C07229=1051.943,291.102,-104.776,172.563,37.718,157.135
C07230=1051.936,290.839,-104.743,172.560,37.714,157.134
C07231=1051.929,290.577,-104.709,172.556,37.711,157.134
C07232=1051.922,290.315,-104.675,172.553,37.708,157.133
C07233=1051.916,290.053,-104.642,172.550,37.704,157.132
C07234=1051.909,289.805,-104.611,172.546,37.701,157.131
C07235=1051.902,289.557,-104.579,172.544,37.697,157.130
C07236=1051.896,289.309,-104.547,172.540,37.694,157.130
C07237=1051.889,289.061,-104.516,172.537,37.690,157.129
C07238=1051.883,288.813,-104.484,172.534,37.687,157.128
C07239=1051.876,288.565,-104.451,172.530,37.683,157.127
C07240=1051.870,288.317,-104.420,172.528,37.680,157.126
C07241=1051.863,288.069,-104.389,172.524,37.677,157.126
C07242=1051.857,287.822,-104.358,172.522,37.673,157.125
C07243=1051.850,287.574,-104.327,172.518,37.670,157.124
C07244=1051.844,287.326,-104.295,172.516,37.667,157.123
C07245=1051.837,287.078,-104.264,172.512,37.663,157.123
C07246=1051.831,286.830,-104.232,172.509,37.660,157.122
C07247=1051.824,286.582,-104.200,172.506,37.657,157.121
C07248=1051.817,286.334,-104.169,172.503,37.653,157.120
C07249=1051.811,286.086,-104.138,172.500,37.650,157.119
C07250=1051.804,285.838,-104.106,172.497,37.647,157.119
C07251=1051.798,285.590,-104.076,172.493,37.643,157.118
C07252=1051.791,285.342,-104.044,172.491,37.640,157.117
C07253=1051.785,285.095,-104.013,172.487,37.637,157.116
C07254=1051.778,284.847,-103.982,172.485,37.634,157.116
C07255=1051.771,284.599,-103.950,172.481,37.630,157.115
C07256=1051.765,284.350,-103.919,172.479,37.627,157.114
C07257=1051.759,284.103,-103.888,172.475,37.623,157.113
C07258=1051.752,283.855,-103.857,172.472,37.620,157.113
C07259=1051.746,283.607,-103.826,172.469,37.617,157.112
C07260=1051.739,283.359,-103.795,172.466,37.613,157.111
C07261=1051.733,283.111,-103.764,172.463,37.610,157.110
C07262=1051.726,282.864,-103.732,172.460,37.606,157.109
C07263=1051.720,282.615,-103.702,172.458,37.604,157.109
C07264=1051.713,282.367,-103.670,172.454,37.600,157.108
C07265=1051.707,282.119,-103.640,172.451,37.597,157.107
C07266=1051.700,281.871,-103.608,172.448,37.593,157.106
C07267=1051.694,281.624,-103.577,172.445,37.590,157.106
C07268=1051.687,281.375,-103.546,172.442,37.587,157.105
C07269=1051.681,281.128,-103.515,172.439,37.583,157.104
C07270=1051.675,280.879,-103.484,172.437,37.580,157.103
C07271=1051.668,280.631,-103.453,172.433,37.576,157.103
C07272=1051.661,280.383,-103.422,172.430,37.574,157.102
C07273=1051.655,280.136,-103.391,172.427,37.570,157.101
C07274=1051.649,279.888,-103.360,172.424,37.567,157.100
C07275=1051.642,279.639,-103.329,172.421,37.563,157.100
C07276=1051.636,279.392,-103.298,172.418,37.560,157.099
C07277=1051.630,279.143,-103.267,172.416,37.557,157.098
C07278=1051.623,278.895,-103.237,172.412,37.553,157.097
C07279=1051.617,278.648,-103.205,172.410,37.551,157.097
C07280=1051.610,278.400,-103.175,172.406,37.547,157.096
C07281=1051.604,278.151,-103.145,172.403,37.544,157.095
C07282=1051.597,277.904,-103.114,172.401,37.541,157.094
C07283=1051.591,277.655,-103.083,172.397,37.537,157.094
C07284=1051.584,277.407,-103.051,172.395,37.534,157.093
C07285=1051.578,277.160,-103.022,172.391,37.531,157.092
C07286=1051.571,276.909,-102.990,172.389,37.527,157.091
C07287=1051.565,276.657,-102.960,172.386,37.524,157.091
C07288=1051.558,276.407,-102.928,172.382,37.520,157.090
C07289=1051.551,276.156,-102.898,172.380,37.518,157.089
C07290=1051.545,275.908,-102.867,172.377,37.514,157.088
C07291=1051.539,275.660,-102.836,172.374,37.511,157.088
C07292=1051.533,275.412,-102.805,172.371,37.508,157.087
C07293=1051.526,275.164,-102.775,172.368,37.504,157.086
C07294=1051.519,274.916,-102.745,172.365,37.501,157.085
C07295=1051.513,274.668,-102.714,172.363,37.498,157.085
C07296=1051.507,274.419,-102.684,172.359,37.494,157.084
C07297=1051.500,274.172,-102.653,172.357,37.491,157.083
C07298=1051.494,273.924,-102.622,172.354,37.488,157.082
C07299=1051.487,273.675,-102.592,172.350,37.485,157.082
C07300=1051.481,273.428,-102.562,172.348,37.482,157.081
C07301=1051.474,273.179,-102.531,172.345,37.478,157.080
C07302=1051.468,272.932,-102.501,172.342,37.475,157.079
C07303=1051.461,272.683,-102.471,172.339,37.472,157.079
C07304=1051.455,272.436,-102.440,172.337,37.468,157.078
C07305=1051.449,272.187,-102.410,172.333,37.465,157.077
C07306=1051.442,271.939,-102.380,172.331,37.462,157.077
C07307=1051.436,271.691,-102.349,172.328,37.458,157.076
C07308=1051.429,271.443,-102.319,172.325,37.456,157.075
C07309=1051.423,271.195,-102.289,172.322,37.452,157.074
C07310=1051.416,270.947,-102.259,172.320,37.449,157.074
C07311=1051.410,270.699,-102.228,172.317,37.446,157.073
C07312=1051.403,270.451,-102.198,172.313,37.442,157.072
C07313=1051.397,270.203,-102.168,172.311,37.439,157.071
C07314=1051.390,269.955,-102.138,172.308,37.436,157.071
C07315=1051.384,269.707,-102.107,172.305,37.433,157.070
C07316=1051.377,269.459,-102.077,172.302,37.429,157.069
C07317=1051.371,269.210,-102.048,172.300,37.427,157.069
C07318=1051.364,268.962,-102.017,172.297,37.423,157.068
C07319=1051.358,268.714,-101.987,172.294,37.420,157.067
C07320=1051.352,268.467,-101.957,172.291,37.417,157.066
C07321=1051.346,268.218,-101.927,172.289,37.413,157.066
C07322=1051.339,267.970,-101.898,172.285,37.410,157.065
C07323=1051.332,267.722,-101.867,172.283,37.407,157.064
C07324=1051.326,267.474,-101.837,172.280,37.404,157.064
C07325=1051.319,267.226,-101.807,172.278,37.400,157.063
C07326=1051.314,266.977,-101.777,172.274,37.398,157.062
C07327=1051.306,266.729,-101.747,172.272,37.394,157.061
C07328=1051.300,266.482,-101.717,172.269,37.391,157.061
C07329=1051.294,266.232,-101.687,172.267,37.388,157.060
C07330=1051.287,265.985,-101.658,172.263,37.385,157.059
C07331=1051.281,265.737,-101.628,172.261,37.381,157.058
C07332=1051.275,265.488,-101.598,172.258,37.378,157.058
C07333=1051.268,265.241,-101.568,172.256,37.375,157.057
C07334=1051.261,264.993,-101.538,172.252,37.372,157.056
C07335=1051.255,264.744,-101.508,172.250,37.368,157.056
C07336=1051.249,264.497,-101.479,172.247,37.365,157.055
C07337=1051.242,264.248,-101.449,172.244,37.362,157.054
C07338=1051.236,264.001,-101.420,172.242,37.359,157.053
C07339=1051.229,263.753,-101.390,172.238,37.356,157.053
C07340=1051.223,263.506,-101.360,172.236,37.352,157.052
C07341=1051.216,263.258,-101.331,172.233,37.349,157.051
C07342=1051.210,263.012,-101.301,172.231,37.346,157.050
C07343=1051.204,262.764,-101.271,172.228,37.343,157.050
C07344=1051.197,262.517,-101.242,172.225,37.340,157.049
C07345=1051.191,262.269,-101.212,172.222,37.336,157.048
C07346=1051.184,262.021,-101.183,172.220,37.333,157.048
C07347=1051.178,261.772,-101.154,172.217,37.330,157.047
C07348=1051.171,261.525,-101.124,172.215,37.327,157.046
C07349=1051.165,261.277,-101.095,172.211,37.324,157.046
C07350=1051.158,261.028,-101.065,172.209,37.321,157.045
C07351=1051.151,260.780,-101.036,172.206,37.318,157.044
C07352=1051.145,260.532,-101.007,172.204,37.315,157.044
C07353=1051.138,260.283,-100.977,172.201,37.311,157.043
C07354=1051.132,260.036,-100.947,172.198,37.308,157.042
C07355=1051.125,259.787,-100.918,172.196,37.305,157.042
C07356=1051.119,259.539,-100.889,172.193,37.302,157.041
C07357=1051.112,259.291,-100.859,172.191,37.299,157.040
C07358=1051.105,259.042,-100.830,172.188,37.295,157.039
C07359=1051.099,258.794,-100.801,172.184,37.293,157.039
C07360=1051.093,258.546,-100.772,172.182,37.290,157.038
C07361=1051.086,258.298,-100.743,172.179,37.286,157.037
C07362=1051.079,258.050,-100.713,172.177,37.283,157.037
C07363=1051.072,257.802,-100.684,172.175,37.280,157.036
C07364=1051.066,257.554,-100.655,172.172,37.277,157.035
C07365=1051.059,257.305,-100.626,172.170,37.274,157.035
C07366=1051.053,257.057,-100.597,172.166,37.270,157.034
C07367=1051.047,256.809,-100.568,172.164,37.267,157.033
C07368=1051.040,256.561,-100.538,172.161,37.264,157.032
C07369=1051.033,256.312,-100.508,172.159,37.261,157.032
C07370=1051.027,256.064,-100.479,172.156,37.258,157.031
C07371=1051.021,255.816,-100.450,172.154,37.255,157.030
C07372=1051.015,255.568,-100.421,172.151,37.252,157.030
C07373=1051.008,255.319,-100.392,172.148,37.249,157.029
C07374=1051.001,255.071,-100.363,172.145,37.245,157.028
C07375=1050.995,254.823,-100.334,172.143,37.242,157.028
C07376=1050.988,254.575,-100.305,172.140,37.239,157.027
C07377=1050.982,254.327,-100.276,172.138,37.236,157.026
C07378=1050.976,254.093,-100.249,172.135,37.233,157.026
C07379=1050.970,253.860,-100.221,172.133,37.230,157.025
C07380=1050.964,253.626,-100.194,172.130,37.227,157.024
C07381=1050.958,253.392,-100.167,172.128,37.223,157.023
C07382=1050.952,253.158,-100.139,172.125,37.221,157.023
C07383=1050.946,252.925,-100.112,172.123,37.218,157.022
C07384=1050.940,252.692,-100.085,172.120,37.215,157.022
C07385=1050.934,252.458,-100.057,172.118,37.212,157.021
C07386=1050.928,252.210,-100.028,172.116,37.209,157.020
C07387=1050.920,251.962,-99.999,172.113,37.205,157.019
C07388=1050.914,251.713,-99.971,172.111,37.202,157.019
C07389=1050.908,251.465,-99.942,172.108,37.199,157.018
C07390=1050.902,251.217,-99.913,172.106,37.196,157.017
C07391=1050.896,250.969,-99.884,172.103,37.192,157.017
C07392=1050.889,250.720,-99.855,172.101,37.189,157.016
C07393=1050.883,250.472,-99.826,172.098,37.186,157.015
C07394=1050.877,250.224,-99.797,172.096,37.183,157.015
C07395=1050.871,249.975,-99.768,172.093,37.180,157.014
C07396=1050.864,249.728,-99.740,172.091,37.176,157.013
C07397=1050.858,249.479,-99.711,172.088,37.174,157.013
C07398=1050.851,249.201,-99.678,172.085,37.169,157.012
C07399=1050.843,248.924,-99.646,172.082,37.166,157.011
C07400=1050.837,248.646,-99.614,172.079,37.162,157.010
C07401=1050.830,248.368,-99.582,172.077,37.159,157.009
C07402=1050.823,248.121,-99.553,172.075,37.156,157.009
C07403=1050.817,247.872,-99.525,172.072,37.152,157.008
C07404=1050.810,247.624,-99.496,172.070,37.149,157.007
C07405=1050.804,247.376,-99.467,172.067,37.146,157.006
C07406=1050.798,247.127,-99.438,172.065,37.143,157.006
C07407=1050.792,246.879,-99.409,172.062,37.139,157.005
C07408=1050.786,246.631,-99.380,172.060,37.136,157.004
C07409=1050.779,246.382,-99.353,172.057,37.133,157.004
C07410=1050.773,246.134,-99.323,172.055,37.130,157.003
C07411=1050.767,245.886,-99.294,172.052,37.126,157.002
C07412=1050.761,245.637,-99.266,172.050,37.123,157.002
C07413=1050.754,245.389,-99.238,172.047,37.120,157.001
C07414=1050.748,245.141,-99.209,172.045,37.117,157.000
C07415=1050.741,244.892,-99.180,172.042,37.114,157.000
C07416=1050.735,244.644,-99.153,172.040,37.111,156.999
C07417=1050.729,244.396,-99.124,172.037,37.108,156.998
C07418=1050.722,244.147,-99.096,172.035,37.104,156.997
C07419=1050.716,243.899,-99.067,172.032,37.101,156.997
C07420=1050.710,243.651,-99.038,172.030,37.098,156.996
C07421=1050.703,243.403,-99.010,172.027,37.095,156.995
C07422=1050.697,243.155,-98.982,172.025,37.092,156.995
C07423=1050.690,242.907,-98.954,172.022,37.088,156.994
C07424=1050.684,242.658,-98.925,172.020,37.085,156.993
C07425=1050.678,242.409,-98.897,172.017,37.082,156.993
C07426=1050.671,242.162,-98.869,172.015,37.079,156.992
C07427=1050.666,241.913,-98.840,172.013,37.076,156.991
C07428=1050.659,241.665,-98.812,172.010,37.072,156.990
C07429=1050.653,241.416,-98.783,172.008,37.069,156.990
C07430=1050.646,241.168,-98.756,172.005,37.066,156.989
C07431=1050.639,240.920,-98.727,172.003,37.063,156.988
C07432=1050.633,240.671,-98.699,172.000,37.060,156.988
C07433=1050.626,240.423,-98.671,171.999,37.056,156.987
C07434=1050.620,240.174,-98.643,171.996,37.053,156.986
C07435=1050.613,239.926,-98.614,171.994,37.050,156.986
C07436=1050.607,239.678,-98.587,171.991,37.047,156.985
C07437=1050.601,239.429,-98.558,171.989,37.044,156.984
C07438=1050.595,239.181,-98.531,171.987,37.041,156.984
C07439=1050.588,238.933,-98.503,171.984,37.037,156.983
C07440=1050.582,238.685,-98.474,171.982,37.034,156.982
C07441=1050.575,238.436,-98.446,171.979,37.031,156.982
C07442=1050.568,238.188,-98.419,171.977,37.028,156.981
C07443=1050.562,237.939,-98.390,171.974,37.025,156.980
C07444=1050.556,237.691,-98.363,171.972,37.021,156.980
C07445=1050.549,237.442,-98.335,171.969,37.018,156.979
C07446=1050.542,237.194,-98.307,171.968,37.015,156.978
C07447=1050.537,236.946,-98.279,171.965,37.012,156.977
C07448=1050.530,236.698,-98.251,171.963,37.009,156.977
C07449=1050.523,236.449,-98.223,171.961,37.006,156.976
C07450=1050.517,236.201,-98.195,171.958,37.002,156.975
C07451=1050.511,235.952,-98.167,171.956,36.999,156.975
C07452=1050.504,235.704,-98.139,171.953,36.996,156.974
C07453=1050.497,235.455,-98.112,171.951,36.993,156.973
C07454=1050.491,235.201,-98.083,171.948,36.990,156.973
C07455=1050.485,234.947,-98.055,171.946,36.986,156.972
C07456=1050.478,234.694,-98.026,171.944,36.983,156.971
C07457=1050.472,234.439,-97.997,171.942,36.980,156.971
C07458=1050.465,234.191,-97.970,171.939,36.977,156.970
C07459=1050.459,233.943,-97.942,171.937,36.973,156.969
C07460=1050.453,233.694,-97.914,171.934,36.970,156.969
C07461=1050.447,233.446,-97.886,171.932,36.967,156.968
C07462=1050.440,233.198,-97.859,171.930,36.964,156.967
C07463=1050.433,232.949,-97.831,171.928,36.960,156.966
C07464=1050.427,232.700,-97.804,171.926,36.957,156.966
C07465=1050.422,232.452,-97.776,171.923,36.954,156.965
C07466=1050.415,232.204,-97.748,171.921,36.951,156.964
C07467=1050.408,231.955,-97.720,171.918,36.948,156.964
C07468=1050.402,231.707,-97.693,171.916,36.944,156.963
C07469=1050.395,231.458,-97.665,171.913,36.941,156.962
C07470=1050.389,231.211,-97.638,171.912,36.938,156.962
C07471=1050.383,230.962,-97.611,171.909,36.935,156.961
C07472=1050.377,230.713,-97.582,171.907,36.932,156.960
C07473=1050.371,230.465,-97.555,171.904,36.928,156.960
C07474=1050.364,230.217,-97.527,171.902,36.925,156.959
C07475=1050.357,229.968,-97.499,171.901,36.922,156.958
C07476=1050.351,229.719,-97.472,171.898,36.919,156.958
C07477=1050.345,229.471,-97.445,171.896,36.916,156.957
C07478=1050.338,229.223,-97.417,171.893,36.912,156.956
C07479=1050.331,228.974,-97.390,171.891,36.909,156.956
C07480=1050.325,228.725,-97.363,171.889,36.906,156.955
C07481=1050.319,228.478,-97.335,171.887,36.903,156.954
C07482=1050.312,228.229,-97.307,171.885,36.900,156.954
C07483=1050.306,227.980,-97.280,171.882,36.897,156.953
C07484=1050.300,227.732,-97.253,171.880,36.893,156.952
C07485=1050.293,227.483,-97.226,171.877,36.890,156.951
C07486=1050.286,227.235,-97.199,171.876,36.887,156.951
C07487=1050.279,226.987,-97.171,171.873,36.884,156.950
C07488=1050.273,226.738,-97.145,171.871,36.881,156.949
C07489=1050.267,226.490,-97.117,171.868,36.877,156.949
C07490=1050.260,226.241,-97.090,171.867,36.874,156.948
C07491=1050.254,225.993,-97.062,171.865,36.871,156.947
C07492=1050.248,225.745,-97.035,171.862,36.868,156.947
C07493=1050.241,225.496,-97.008,171.860,36.865,156.946
C07494=1050.235,225.248,-96.980,171.857,36.862,156.945
C07495=1050.228,224.999,-96.954,171.856,36.858,156.945
C07496=1050.221,224.751,-96.926,171.853,36.855,156.944
C07497=1050.216,224.502,-96.900,171.851,36.852,156.943
C07498=1050.209,224.254,-96.872,171.848,36.849,156.943
C07499=1050.203,224.006,-96.845,171.847,36.846,156.942
C07500=1050.197,223.757,-96.817,171.845,36.842,156.941
C07501=1050.190,223.508,-96.790,171.842,36.839,156.941
C07502=1050.184,223.260,-96.764,171.840,36.836,156.940
C07503=1050.177,223.012,-96.737,171.838,36.833,156.939
C07504=1050.171,222.763,-96.710,171.836,36.829,156.939
C07505=1050.164,222.515,-96.682,171.833,36.826,156.938
C07506=1050.158,222.266,-96.655,171.831,36.823,156.937
C07507=1050.152,222.018,-96.628,171.830,36.819,156.937
C07508=1050.146,221.769,-96.601,171.827,36.816,156.936
C07509=1050.139,221.521,-96.575,171.825,36.813,156.935
C07510=1050.132,221.259,-96.545,171.823,36.809,156.934
C07511=1050.126,220.997,-96.517,171.821,36.806,156.934
C07512=1050.119,220.736,-96.489,171.818,36.803,156.933
C07513=1050.113,220.474,-96.460,171.816,36.799,156.932
C07514=1050.105,220.226,-96.433,171.813,36.796,156.932
C07515=1050.099,219.977,-96.407,171.812,36.793,156.931
C07516=1050.092,219.729,-96.380,171.809,36.790,156.930
C07517=1050.087,219.480,-96.354,171.807,36.787,156.930
C07518=1050.080,219.232,-96.326,171.806,36.783,156.929
C07519=1050.073,218.984,-96.300,171.803,36.780,156.928
C07520=1050.067,218.735,-96.273,171.801,36.777,156.927
C07521=1050.060,218.486,-96.246,171.798,36.774,156.927
C07522=1050.054,218.238,-96.220,171.797,36.771,156.926
C07523=1050.047,217.989,-96.192,171.794,36.767,156.925
C07524=1050.041,217.741,-96.166,171.792,36.764,156.925
C07525=1050.035,217.492,-96.139,171.791,36.760,156.924
C07526=1050.028,217.244,-96.113,171.788,36.757,156.923
C07527=1050.022,216.995,-96.086,171.786,36.754,156.923
C07528=1050.015,216.747,-96.060,171.784,36.751,156.922
C07529=1050.009,216.498,-96.033,171.782,36.748,156.921
C07530=1050.003,216.250,-96.005,171.779,36.744,156.921
C07531=1049.996,216.001,-95.979,171.778,36.741,156.920
C07532=1049.990,215.753,-95.952,171.776,36.738,156.919
C07533=1049.983,215.504,-95.926,171.773,36.735,156.919
C07534=1049.977,215.256,-95.899,171.772,36.731,156.918
C07535=1049.970,215.007,-95.873,171.769,36.728,156.917
C07536=1049.964,214.759,-95.846,171.767,36.725,156.917
C07537=1049.958,214.510,-95.820,171.765,36.722,156.916
C07538=1049.951,214.262,-95.793,171.763,36.719,156.915
C07539=1049.945,214.013,-95.767,171.761,36.715,156.915
C07540=1049.938,213.765,-95.740,171.759,36.712,156.914
C07541=1049.932,213.516,-95.713,171.757,36.708,156.913
C07542=1049.925,213.267,-95.687,171.755,36.705,156.913
C07543=1049.920,213.019,-95.660,171.753,36.702,156.912
C07544=1049.913,212.771,-95.634,171.750,36.699,156.911
C07545=1049.907,212.522,-95.607,171.749,36.695,156.910
C07546=1049.900,212.274,-95.581,171.747,36.692,156.910
C07547=1049.894,212.025,-95.554,171.744,36.689,156.909
C07548=1049.887,211.777,-95.528,171.743,36.686,156.908
C07549=1049.881,211.528,-95.501,171.740,36.682,156.908
C07550=1049.874,211.280,-95.475,171.739,36.679,156.907
C07551=1049.868,211.031,-95.450,171.736,36.675,156.906
C07552=1049.862,210.782,-95.423,171.734,36.672,156.906
C07553=1049.855,210.534,-95.397,171.733,36.669,156.905
C07554=1049.849,210.285,-95.370,171.730,36.666,156.904
C07555=1049.842,210.037,-95.344,171.729,36.662,156.904
C07556=1049.836,209.789,-95.318,171.726,36.659,156.903
C07557=1049.830,209.539,-95.291,171.724,36.656,156.902
C07558=1049.823,209.291,-95.265,171.723,36.653,156.902
C07559=1049.817,209.043,-95.239,171.720,36.649,156.901
C07560=1049.810,208.794,-95.212,171.719,36.646,156.900
C07561=1049.804,208.546,-95.186,171.716,36.643,156.899
C07562=1049.797,208.297,-95.160,171.714,36.640,156.899
C07563=1049.791,208.049,-95.134,171.712,36.636,156.898
C07564=1049.785,207.800,-95.108,171.710,36.633,156.897
C07565=1049.778,207.551,-95.081,171.709,36.629,156.897
C07566=1049.771,207.295,-95.055,171.706,36.626,156.896
C07567=1049.765,207.039,-95.028,171.704,36.623,156.895
C07568=1049.758,206.783,-95.001,171.702,36.619,156.895
C07569=1049.752,206.527,-94.974,171.700,36.616,156.894
C07570=1049.726,205.475,-94.869,171.467,36.519,156.874
C07571=1049.720,205.226,-94.843,171.464,36.516,156.873
C07572=1049.714,204.977,-94.818,171.462,36.514,156.873
C07573=1049.707,204.729,-94.793,171.460,36.512,156.872
C07574=1049.702,204.480,-94.768,171.457,36.509,156.872
C07575=1049.695,204.232,-94.744,171.454,36.507,156.871
C07576=1049.689,203.983,-94.718,171.452,36.504,156.871
C07577=1049.683,203.734,-94.694,171.449,36.501,156.870
C07578=1049.677,203.485,-94.668,171.446,36.499,156.870
C07579=1049.671,203.237,-94.643,171.444,36.497,156.869
C07580=1049.665,202.988,-94.619,171.442,36.494,156.869
C07581=1049.659,202.739,-94.593,171.438,36.492,156.868
C07582=1049.654,202.491,-94.568,171.436,36.489,156.868
C07583=1049.648,202.242,-94.544,171.434,36.487,156.867
C07584=1049.641,201.993,-94.518,171.431,36.484,156.867
C07585=1049.636,201.744,-94.494,171.428,36.482,156.866
C07586=1049.629,201.496,-94.469,171.426,36.480,156.866
C07587=1049.623,201.247,-94.445,171.424,36.477,156.865
C07588=1049.617,200.998,-94.419,171.420,36.475,156.865
C07589=1049.610,200.749,-94.395,171.418,36.472,156.864
C07590=1049.604,200.501,-94.370,171.416,36.470,156.864
C07591=1049.599,200.252,-94.346,171.413,36.467,156.863
C07592=1049.592,200.004,-94.321,171.410,36.465,156.863
C07593=1049.586,199.755,-94.296,171.408,36.463,156.862
C07594=1049.579,199.506,-94.272,171.406,36.460,156.862
C07595=1049.574,199.258,-94.247,171.403,36.458,156.861
C07596=1049.567,199.009,-94.223,171.400,36.456,156.861
C07597=1049.561,198.760,-94.198,171.398,36.454,156.861
C07598=1049.556,198.511,-94.174,171.396,36.451,156.860
C07599=1049.549,198.263,-94.149,171.392,36.449,156.860
C07600=1049.543,198.014,-94.125,171.390,36.446,156.859
C07601=1049.537,197.765,-94.101,171.388,36.444,156.859
C07602=1049.531,197.517,-94.076,171.385,36.441,156.858
C07603=1049.525,197.267,-94.051,171.383,36.439,156.858
C07604=1049.518,197.018,-94.027,171.380,36.437,156.857
C07605=1049.512,196.771,-94.002,171.378,36.435,156.857
C07606=1049.506,196.522,-93.978,171.375,36.432,156.856
C07607=1049.501,196.273,-93.954,171.373,36.430,156.856
C07608=1049.494,196.025,-93.929,171.370,36.427,156.855
C07609=1049.488,195.775,-93.904,171.367,36.425,156.855
C07610=1049.482,195.527,-93.881,171.365,36.423,156.854
C07611=1049.476,195.278,-93.856,171.363,36.421,156.854
C07612=1049.470,195.029,-93.831,171.361,36.418,156.853
C07613=1049.464,194.781,-93.807,171.357,36.416,156.853
C07614=1049.458,194.532,-93.782,171.355,36.413,156.852
C07615=1049.452,194.283,-93.759,171.353,36.411,156.852
C07616=1049.446,194.034,-93.734,171.351,36.409,156.851
C07617=1049.439,193.786,-93.709,171.348,36.407,156.851
C07618=1049.433,193.537,-93.685,171.345,36.404,156.851
C07619=1049.427,193.288,-93.661,171.343,36.402,156.850
C07620=1049.422,193.039,-93.637,171.340,36.399,156.850
C07621=1049.415,192.790,-93.613,171.338,36.397,156.849
C07622=1049.410,192.542,-93.588,171.336,36.395,156.849
C07623=1049.403,192.293,-93.564,171.333,36.393,156.848
C07624=1049.397,192.044,-93.539,171.330,36.390,156.848
C07625=1049.391,191.796,-93.515,171.328,36.388,156.847
C07626=1049.385,191.547,-93.491,171.326,36.385,156.847
C07627=1049.379,191.298,-93.467,171.324,36.384,156.846
C07628=1049.373,191.049,-93.443,171.321,36.381,156.846
C07629=1049.368,190.801,-93.418,171.318,36.379,156.846
C07630=1049.361,190.552,-93.394,171.316,36.376,156.845
C07631=1049.354,190.267,-93.367,171.314,36.374,156.845
C07632=1049.347,189.983,-93.339,171.310,36.371,156.844
C07633=1049.341,189.699,-93.312,171.308,36.368,156.843
C07634=1049.334,189.414,-93.284,171.305,36.366,156.843
C07635=1049.328,189.166,-93.260,171.302,36.364,156.842
C07636=1049.322,188.917,-93.235,171.300,36.361,156.842
C07637=1049.316,188.669,-93.212,171.298,36.359,156.842
C07638=1049.310,188.419,-93.187,171.296,36.357,156.841
C07639=1049.304,188.171,-93.163,171.293,36.354,156.841
C07640=1049.299,187.921,-93.139,171.291,36.352,156.840
C07641=1049.292,187.673,-93.116,171.289,36.350,156.840
C07642=1049.287,187.424,-93.091,171.286,36.348,156.839
C07643=1049.281,187.175,-93.067,171.283,36.345,156.839
C07644=1049.275,186.927,-93.043,171.281,36.343,156.838
C07645=1049.269,186.678,-93.019,171.279,36.340,156.838
C07646=1049.263,186.429,-92.995,171.276,36.339,156.837
C07647=1049.257,186.180,-92.971,171.274,36.336,156.837
C07648=1049.251,185.932,-92.947,171.272,36.334,156.836
C07649=1049.246,185.683,-92.924,171.270,36.331,156.836
C07650=1049.239,185.434,-92.900,171.267,36.329,156.836
C07651=1049.234,185.185,-92.875,171.264,36.327,156.835
C07652=1049.228,184.937,-92.852,171.262,36.324,156.835
C07653=1049.222,184.688,-92.827,171.260,36.322,156.834
C07654=1049.216,184.439,-92.803,171.257,36.320,156.834
C07655=1049.211,184.190,-92.780,171.255,36.318,156.833
C07656=1049.204,183.941,-92.756,171.253,36.315,156.833
C07657=1049.198,183.693,-92.732,171.251,36.313,156.832
C07658=1049.192,183.443,-92.709,171.248,36.311,156.832
C07659=1049.186,183.195,-92.685,171.246,36.309,156.832
C07660=1049.179,182.946,-92.661,171.244,36.307,156.831
C07661=1049.173,182.697,-92.638,171.241,36.305,156.831
C07662=1049.167,182.448,-92.614,171.238,36.303,156.830
C07663=1049.161,182.199,-92.591,171.236,36.301,156.830
C07664=1049.155,181.951,-92.568,171.234,36.299,156.830
C07665=1049.148,181.702,-92.544,171.232,36.296,156.829
C07666=1049.143,181.453,-92.521,171.230,36.295,156.829
C07667=1049.135,181.204,-92.497,171.227,36.292,156.828
C07668=1049.129,180.956,-92.474,171.225,36.290,156.828
C07669=1049.123,180.707,-92.450,171.223,36.288,156.828
C07670=1049.117,180.458,-92.427,171.220,36.286,156.827
C07671=1049.111,180.209,-92.404,171.217,36.284,156.827
C07672=1049.105,179.960,-92.380,171.215,36.282,156.826
C07673=1049.099,179.711,-92.357,171.213,36.280,156.826
C07674=1049.093,179.463,-92.334,171.211,36.277,156.825
C07675=1049.086,179.214,-92.310,171.208,36.276,156.825
C07676=1049.081,178.965,-92.287,171.206,36.274,156.825
C07677=1049.074,178.716,-92.263,171.204,36.271,156.824
C07678=1049.068,178.467,-92.240,171.202,36.269,156.824
C07679=1049.062,178.219,-92.216,171.199,36.267,156.823
C07680=1049.055,177.969,-92.193,171.197,36.265,156.823
C07681=1049.049,177.720,-92.170,171.195,36.263,156.822
C07682=1049.043,177.472,-92.147,171.192,36.261,156.822
C07683=1049.038,177.223,-92.124,171.190,36.259,156.822
C07684=1049.031,176.974,-92.100,171.187,36.257,156.821
C07685=1049.025,176.725,-92.077,171.185,36.255,156.821
C07686=1049.020,176.476,-92.054,171.183,36.252,156.820
C07687=1049.013,176.227,-92.030,171.181,36.250,156.820
C07688=1049.007,175.979,-92.007,171.178,36.249,156.820
C07689=1049.000,175.731,-91.984,171.176,36.246,156.819
C07690=1048.994,175.481,-91.961,171.174,36.244,156.819
C07691=1048.988,175.232,-91.938,171.172,36.242,156.818
C07692=1048.983,174.983,-91.915,171.170,36.240,156.818
C07693=1048.977,174.735,-91.891,171.167,36.238,156.818
C07694=1048.970,174.485,-91.868,171.165,36.236,156.817
C07695=1048.963,174.201,-91.842,171.163,36.233,156.817
C07696=1048.956,173.916,-91.815,171.160,36.231,156.816
C07697=1048.950,173.631,-91.788,171.157,36.229,156.816
C07698=1048.942,173.347,-91.762,171.155,36.226,156.815
C07699=1048.937,173.098,-91.739,171.153,36.224,156.815
C07700=1048.931,172.849,-91.716,171.151,36.222,156.814
C07701=1048.925,172.600,-91.693,171.148,36.220,156.814
C07702=1048.918,172.351,-91.669,171.146,36.218,156.814
C07703=1048.912,172.102,-91.646,171.144,36.216,156.813
C07704=1048.906,171.854,-91.623,171.142,36.214,156.813
C07705=1048.901,171.605,-91.601,171.139,36.212,156.812
C07706=1048.895,171.356,-91.578,171.137,36.210,156.812
C07707=1048.889,171.107,-91.555,171.135,36.207,156.812
C07708=1048.882,170.858,-91.531,171.133,36.206,156.811
C07709=1048.876,170.609,-91.508,171.131,36.203,156.811
C07710=1048.870,170.360,-91.485,171.128,36.201,156.810
C07711=1048.865,170.112,-91.462,171.126,36.199,156.810
C07712=1048.859,169.863,-91.439,171.124,36.197,156.810
C07713=1048.853,169.614,-91.416,171.122,36.195,156.809
C07714=1048.847,169.365,-91.394,171.119,36.193,156.809
C07715=1048.840,169.116,-91.371,171.117,36.191,156.808
C07716=1048.834,168.867,-91.347,171.115,36.189,156.808
C07717=1048.829,168.618,-91.324,171.113,36.187,156.807
C07718=1048.823,168.369,-91.301,171.111,36.185,156.807
C07719=1048.817,168.121,-91.278,171.108,36.183,156.807
C07720=1048.811,167.872,-91.255,171.106,36.180,156.806
C07721=1048.805,167.623,-91.233,171.104,36.179,156.806
C07722=1048.799,167.374,-91.210,171.102,36.176,156.805
C07723=1048.793,167.125,-91.187,171.099,36.174,156.805
C07724=1048.788,166.876,-91.164,171.097,36.172,156.805
C07725=1048.782,166.627,-91.141,171.095,36.170,156.804
C07726=1048.775,166.379,-91.119,171.093,36.168,156.804
C07727=1048.769,166.129,-91.096,171.091,36.166,156.804
C07728=1048.763,165.880,-91.073,171.088,36.164,156.803
C07729=1048.758,165.632,-91.050,171.086,36.162,156.803
C07730=1048.752,165.383,-91.027,171.084,36.159,156.802
C07731=1048.745,165.134,-91.004,171.082,36.158,156.802
C07732=1048.740,164.885,-90.981,171.079,36.156,156.801
C07733=1048.734,164.636,-90.959,171.077,36.153,156.801
C07734=1048.729,164.387,-90.936,171.076,36.151,156.801
C07735=1048.723,164.138,-90.913,171.074,36.150,156.800
C07736=1048.716,163.889,-90.891,171.072,36.147,156.800
C07737=1048.711,163.640,-90.868,171.069,36.145,156.799
C07738=1048.705,163.391,-90.845,171.067,36.143,156.799
C07739=1048.699,163.143,-90.822,171.065,36.141,156.799
C07740=1048.693,162.894,-90.800,171.063,36.139,156.798
C07741=1048.687,162.644,-90.778,171.060,36.137,156.798
C07742=1048.682,162.396,-90.755,171.058,36.135,156.797
C07743=1048.676,162.147,-90.732,171.056,36.133,156.797
C07744=1048.669,161.898,-90.709,171.054,36.130,156.797
C07745=1048.664,161.650,-90.687,171.053,36.129,156.796
C07746=1048.658,161.401,-90.664,171.050,36.127,156.796
C07747=1048.653,161.151,-90.642,171.048,36.124,156.795
C07748=1048.647,160.903,-90.619,171.046,36.122,156.795
C07749=1048.641,160.654,-90.596,171.044,36.120,156.795
C07750=1048.635,160.405,-90.573,171.042,36.118,156.794
C07751=1048.629,160.156,-90.552,171.039,36.116,156.794
C07752=1048.623,159.907,-90.529,171.037,36.114,156.793
C07753=1048.617,159.658,-90.506,171.035,36.113,156.793
C07754=1048.611,159.409,-90.485,171.033,36.111,156.793
C07755=1048.605,159.160,-90.462,171.031,36.108,156.792
C07756=1048.599,158.911,-90.440,171.028,36.106,156.792
C07757=1048.593,158.662,-90.417,171.027,36.105,156.792
C07758=1048.587,158.414,-90.395,171.025,36.103,156.791
C07759=1048.579,158.128,-90.370,171.022,36.100,156.791
C07760=1048.572,157.843,-90.344,171.020,36.098,156.790
C07761=1048.565,157.558,-90.319,171.017,36.096,156.790
C07762=1048.559,157.272,-90.294,171.015,36.094,156.790
C07763=1048.553,157.024,-90.271,171.013,36.092,156.789
C07764=1048.547,156.774,-90.249,171.011,36.090,156.789
C07765=1048.541,156.525,-90.226,171.008,36.088,156.788
C07766=1048.535,156.277,-90.204,171.006,36.086,156.788
C07767=1048.528,156.028,-90.182,171.004,36.084,156.788
C07768=1048.523,155.779,-90.159,171.003,36.082,156.787
C07769=1048.517,155.530,-90.137,171.001,36.080,156.787
C07770=1048.510,155.281,-90.115,170.998,36.078,156.786
C07771=1048.505,155.031,-90.093,170.996,36.076,156.786
C07772=1048.498,154.783,-90.071,170.994,36.074,156.786
C07773=1048.492,154.534,-90.049,170.992,36.072,156.785
C07774=1048.486,154.285,-90.026,170.990,36.070,156.785
C07775=1048.481,154.036,-90.005,170.987,36.069,156.785
C07776=1048.475,153.787,-89.983,170.985,36.067,156.784
C07777=1048.468,153.539,-89.961,170.984,36.064,156.784
C07778=1048.462,153.289,-89.939,170.982,36.062,156.783
C07779=1048.456,153.040,-89.916,170.980,36.061,156.783
C07780=1048.450,152.791,-89.894,170.977,36.059,156.783
C07781=1048.444,152.542,-89.873,170.975,36.057,156.782
C07782=1048.437,152.293,-89.851,170.973,36.055,156.782
C07783=1048.432,152.044,-89.828,170.971,36.053,156.782
C07784=1048.426,151.795,-89.807,170.969,36.051,156.781
C07785=1048.420,151.547,-89.785,170.968,36.049,156.781
C07786=1048.414,151.298,-89.763,170.965,36.048,156.781
C07787=1048.408,151.048,-89.741,170.963,36.046,156.780
C07788=1048.402,150.799,-89.718,170.961,36.043,156.780
C07789=1048.396,150.550,-89.697,170.959,36.041,156.779
C07790=1048.390,150.301,-89.675,170.957,36.039,156.779
C07791=1048.384,150.053,-89.653,170.954,36.038,156.779
C07792=1048.378,149.804,-89.632,170.953,36.036,156.778
C07793=1048.372,149.554,-89.609,170.951,36.034,156.778
C07794=1048.366,149.306,-89.587,170.949,36.032,156.778
C07795=1048.359,149.057,-89.565,170.947,36.030,156.777
C07796=1048.354,148.808,-89.544,170.944,36.028,156.777
C07797=1048.348,148.559,-89.522,170.942,36.026,156.777
C07798=1048.342,148.310,-89.501,170.941,36.025,156.776
C07799=1048.335,148.061,-89.478,170.939,36.023,156.776
C07800=1048.329,147.812,-89.457,170.937,36.021,156.775
C07801=1048.324,147.562,-89.435,170.935,36.019,156.775
C07802=1048.318,147.314,-89.413,170.932,36.017,156.775
C07803=1048.312,147.065,-89.392,170.930,36.015,156.774
C07804=1048.305,146.816,-89.369,170.928,36.013,156.774
C07805=1048.299,146.567,-89.348,170.927,36.012,156.774
C07806=1048.293,146.318,-89.326,170.925,36.010,156.773
C07807=1048.287,146.069,-89.305,170.922,36.008,156.773
C07808=1048.281,145.820,-89.284,170.920,36.006,156.773
C07809=1048.274,145.571,-89.262,170.918,36.004,156.772
C07810=1048.268,145.322,-89.240,170.916,36.002,156.772
C07811=1048.262,145.073,-89.219,170.915,36.000,156.772
C07812=1048.257,144.824,-89.198,170.913,35.998,156.771
C07813=1048.250,144.575,-89.176,170.910,35.997,156.771
C07814=1048.244,144.326,-89.154,170.908,35.995,156.771
C07815=1048.238,144.077,-89.133,170.906,35.993,156.770
C07816=1048.232,143.829,-89.111,170.904,35.991,156.770
C07817=1048.226,143.580,-89.089,170.903,35.989,156.769
C07818=1048.220,143.330,-89.067,170.900,35.987,156.769
C07819=1048.214,143.081,-89.046,170.898,35.985,156.769
C07820=1048.208,142.833,-89.024,170.896,35.984,156.768
C07821=1048.202,142.583,-89.003,170.894,35.982,156.768
C07822=1048.196,142.334,-88.981,170.893,35.980,156.768
C07823=1048.189,142.049,-88.958,170.889,35.977,156.767
C07824=1048.182,141.763,-88.932,170.887,35.975,156.767
C07825=1048.175,141.477,-88.908,170.885,35.974,156.766
C07826=1048.168,141.193,-88.884,170.883,35.971,156.766
C07827=1048.162,140.943,-88.862,170.881,35.969,156.766
C07828=1048.156,140.694,-88.840,170.879,35.967,156.765
C07829=1048.150,140.446,-88.819,170.877,35.966,156.765
C07830=1048.144,140.196,-88.797,170.875,35.964,156.765
C07831=1048.138,139.947,-88.777,170.873,35.962,156.764
C07832=1048.133,139.698,-88.755,170.872,35.960,156.764
C07833=1048.126,139.449,-88.734,170.870,35.958,156.764
C07834=1048.120,139.200,-88.712,170.867,35.956,156.763
C07835=1048.113,138.951,-88.691,170.865,35.954,156.763
C07836=1048.108,138.702,-88.670,170.863,35.952,156.762
C07837=1048.102,138.453,-88.648,170.862,35.951,156.762
C07838=1048.096,138.203,-88.627,170.860,35.949,156.762
C07839=1048.089,137.955,-88.606,170.858,35.947,156.762
C07840=1048.083,137.706,-88.585,170.855,35.946,156.761
C07841=1048.077,137.457,-88.563,170.853,35.944,156.761
C07842=1048.072,137.208,-88.542,170.852,35.942,156.760
C07843=1048.065,136.959,-88.522,170.850,35.940,156.760
C07844=1048.059,136.709,-88.500,170.848,35.938,156.760
C07845=1048.053,136.461,-88.479,170.845,35.936,156.759
C07846=1048.047,136.211,-88.458,170.843,35.934,156.759
C07847=1048.040,135.962,-88.437,170.842,35.932,156.759
C07848=1048.035,135.714,-88.415,170.840,35.931,156.758
C07849=1048.029,135.464,-88.394,170.838,35.929,156.758
C07850=1048.023,135.216,-88.374,170.836,35.927,156.758
C07851=1048.017,134.966,-88.352,170.834,35.926,156.757
C07852=1048.010,134.717,-88.331,170.832,35.924,156.757
C07853=1048.004,134.468,-88.311,170.830,35.922,156.757
C07854=1047.998,134.219,-88.289,170.828,35.920,156.756
C07855=1047.992,133.970,-88.267,170.826,35.918,156.756
C07856=1047.986,133.721,-88.247,170.825,35.916,156.756
C07857=1047.980,133.472,-88.226,170.822,35.914,156.755
C07858=1047.974,133.224,-88.204,170.820,35.913,156.755
C07859=1047.968,132.974,-88.184,170.818,35.911,156.755
C07860=1047.962,132.726,-88.163,170.817,35.909,156.754
C07861=1047.956,132.476,-88.141,170.815,35.907,156.754
C07862=1047.949,132.227,-88.121,170.813,35.906,156.754
C07863=1047.944,131.978,-88.100,170.810,35.904,156.753
C07864=1047.938,131.728,-88.079,170.809,35.902,156.753
C07865=1047.932,131.480,-88.058,170.807,35.900,156.753
C07866=1047.926,131.230,-88.037,170.805,35.898,156.752
C07867=1047.919,130.982,-88.016,170.803,35.897,156.752
C07868=1047.914,130.732,-87.996,170.802,35.895,156.752
C07869=1047.907,130.484,-87.975,170.799,35.893,156.751
C07870=1047.901,130.235,-87.955,170.797,35.891,156.751
C07871=1047.895,129.986,-87.933,170.795,35.890,156.751
C07872=1047.888,129.736,-87.913,170.793,35.888,156.750
C07873=1047.883,129.487,-87.891,170.792,35.886,156.750
C07874=1047.876,129.238,-87.871,170.790,35.884,156.750
C07875=1047.870,128.990,-87.850,170.787,35.882,156.749
C07876=1047.864,128.740,-87.829,170.785,35.881,156.749
C07877=1047.857,128.491,-87.808,170.784,35.879,156.749
C07878=1047.851,128.242,-87.788,170.782,35.877,156.748
C07879=1047.845,127.992,-87.767,170.780,35.876,156.748
C07880=1047.839,127.744,-87.747,170.778,35.874,156.748
C07881=1047.832,127.495,-87.726,170.776,35.872,156.747
C07882=1047.827,127.246,-87.705,170.774,35.871,156.747
C07883=1047.820,126.997,-87.685,170.772,35.869,156.747
C07884=1047.815,126.748,-87.664,170.770,35.867,156.746
C07885=1047.808,126.499,-87.643,170.769,35.866,156.746
C07886=1047.801,126.249,-87.623,170.767,35.864,156.746
C07887=1047.794,125.964,-87.599,170.765,35.862,156.745
C07888=1047.787,125.678,-87.576,170.762,35.860,156.745
C07889=1047.781,125.392,-87.553,170.760,35.857,156.745
C07890=1047.773,125.106,-87.529,170.758,35.855,156.744
C07891=1047.768,124.857,-87.508,170.756,35.854,156.744
C07892=1047.761,124.608,-87.487,170.754,35.852,156.744
C07893=1047.755,124.359,-87.467,170.752,35.850,156.743
C07894=1047.749,124.110,-87.447,170.750,35.849,156.743
C07895=1047.743,123.861,-87.426,170.748,35.847,156.743
C07896=1047.737,123.613,-87.406,170.746,35.845,156.742
C07897=1047.731,123.363,-87.385,170.745,35.844,156.742
C07898=1047.725,123.114,-87.365,170.743,35.842,156.742
C07899=1047.718,122.865,-87.344,170.741,35.840,156.741
C07900=1047.713,122.616,-87.323,170.739,35.838,156.741
C07901=1047.706,122.366,-87.303,170.737,35.837,156.741
C07902=1047.700,122.118,-87.283,170.735,35.835,156.740
C07903=1047.694,121.868,-87.262,170.733,35.833,156.740
C07904=1047.688,121.620,-87.241,170.732,35.831,156.740
C07905=1047.682,121.371,-87.221,170.730,35.829,156.739
C07906=1047.676,121.121,-87.200,170.727,35.828,156.739
C07907=1047.670,120.872,-87.180,170.726,35.826,156.739
C07908=1047.663,120.623,-87.160,170.724,35.824,156.738
C07909=1047.658,120.374,-87.139,170.722,35.822,156.738
C07910=1047.652,120.125,-87.119,170.720,35.820,156.738
C07911=1047.645,119.876,-87.099,170.719,35.818,156.737
C07912=1047.639,119.627,-87.079,170.716,35.817,156.737
C07913=1047.633,119.377,-87.058,170.714,35.815,156.737
C07914=1047.627,119.128,-87.038,170.713,35.813,156.736
C07915=1047.621,118.880,-87.018,170.711,35.812,156.736
C07916=1047.616,118.630,-86.997,170.709,35.810,156.736
C07917=1047.609,118.382,-86.976,170.708,35.808,156.736
C07918=1047.603,118.132,-86.956,170.706,35.807,156.735
C07919=1047.597,117.883,-86.935,170.703,35.805,156.735
C07920=1047.591,117.634,-86.915,170.701,35.803,156.734
C07921=1047.585,117.385,-86.895,170.700,35.801,156.734
C07922=1047.579,117.136,-86.875,170.698,35.799,156.734
C07923=1047.574,116.887,-86.854,170.696,35.798,156.734
C07924=1047.567,116.637,-86.834,170.695,35.796,156.733
C07925=1047.561,116.388,-86.814,170.692,35.794,156.733
C07926=1047.555,116.139,-86.794,170.690,35.792,156.732
C07927=1047.549,115.890,-86.773,170.689,35.790,156.732
C07928=1047.543,115.641,-86.753,170.687,35.788,156.732
C07929=1047.537,115.392,-86.733,170.685,35.787,156.732
C07930=1047.532,115.143,-86.713,170.684,35.785,156.731
C07931=1047.525,114.893,-86.692,170.681,35.783,156.731
C07932=1047.519,114.645,-86.673,170.679,35.781,156.731
C07933=1047.513,114.396,-86.653,170.678,35.780,156.730
C07934=1047.507,114.146,-86.632,170.676,35.778,156.730
C07935=1047.501,113.897,-86.612,170.674,35.776,156.730
C07936=1047.495,113.648,-86.592,170.673,35.774,156.729
C07937=1047.489,113.399,-86.571,170.670,35.773,156.729
C07938=1047.483,113.150,-86.551,170.668,35.771,156.729
C07939=1047.477,112.901,-86.531,170.666,35.769,156.728
C07940=1047.471,112.651,-86.512,170.665,35.768,156.728
C07941=1047.465,112.402,-86.492,170.663,35.766,156.728
C07942=1047.459,112.153,-86.472,170.661,35.764,156.727
C07943=1047.453,111.905,-86.452,170.660,35.763,156.727
C07944=1047.446,111.655,-86.432,170.657,35.761,156.727
C07945=1047.440,111.406,-86.412,170.655,35.759,156.726
C07946=1047.434,111.157,-86.392,170.654,35.757,156.726
C07947=1047.428,110.907,-86.372,170.652,35.756,156.726
C07948=1047.422,110.658,-86.352,170.650,35.754,156.725
C07949=1047.416,110.410,-86.332,170.649,35.752,156.725
C07950=1047.409,110.160,-86.312,170.647,35.751,156.725
C07951=1047.402,109.874,-86.290,170.644,35.749,156.724
C07952=1047.395,109.588,-86.267,170.642,35.747,156.724
C07953=1047.388,109.303,-86.244,170.640,35.745,156.724
C07954=1047.381,109.017,-86.221,170.638,35.743,156.723
C07955=1047.375,108.768,-86.201,170.636,35.741,156.723
C07956=1047.369,108.518,-86.182,170.635,35.739,156.723
C07957=1047.363,108.269,-86.162,170.632,35.738,156.723
C07958=1047.356,108.020,-86.142,170.630,35.736,156.722
C07959=1047.350,107.771,-86.123,170.629,35.734,156.722
C07960=1047.344,107.522,-86.103,170.627,35.733,156.722
C07961=1047.338,107.273,-86.083,170.625,35.731,156.721
C07962=1047.332,107.024,-86.063,170.624,35.729,156.721
C07963=1047.326,106.774,-86.044,170.622,35.728,156.721
C07964=1047.320,106.526,-86.024,170.619,35.726,156.720
C07965=1047.313,106.276,-86.005,170.618,35.724,156.720
C07966=1047.307,106.027,-85.985,170.616,35.723,156.720
C07967=1047.301,105.778,-85.965,170.614,35.721,156.719
C07968=1047.295,105.529,-85.946,170.613,35.719,156.719
C07969=1047.289,105.280,-85.926,170.611,35.718,156.719
C07970=1047.283,105.030,-85.905,170.609,35.716,156.718
C07971=1047.276,104.781,-85.887,170.607,35.714,156.718
C07972=1047.270,104.532,-85.867,170.605,35.712,156.718
C07973=1047.265,104.283,-85.847,170.603,35.711,156.718
C07974=1047.259,104.034,-85.827,170.602,35.709,156.717
C07975=1047.252,103.784,-85.808,170.600,35.707,156.717
C07976=1047.246,103.535,-85.788,170.598,35.706,156.717
C07977=1047.239,103.287,-85.769,170.597,35.704,156.716
C07978=1047.234,103.037,-85.749,170.594,35.702,156.716
C07979=1047.228,102.789,-85.729,170.592,35.701,156.716
C07980=1047.222,102.539,-85.710,170.591,35.699,156.715
C07981=1047.216,102.290,-85.690,170.589,35.697,156.715
C07982=1047.209,102.040,-85.671,170.587,35.695,156.715
C07983=1047.203,101.792,-85.651,170.586,35.694,156.714
C07984=1047.197,101.542,-85.632,170.584,35.692,156.714
C07985=1047.191,101.293,-85.612,170.582,35.690,156.714
C07986=1047.186,101.044,-85.593,170.580,35.689,156.713
C07987=1047.179,100.796,-85.573,170.578,35.687,156.713
C07988=1047.173,100.545,-85.554,170.577,35.685,156.713
C07989=1047.167,100.297,-85.534,170.575,35.684,156.713
C07990=1047.160,100.047,-85.515,170.573,35.682,156.712
C07991=1047.155,99.798,-85.496,170.571,35.680,156.712
C07992=1047.148,99.549,-85.477,170.569,35.679,156.712
C07993=1047.142,99.300,-85.457,170.567,35.677,156.711
C07994=1047.136,99.051,-85.437,170.566,35.675,156.711
C07995=1047.129,98.801,-85.418,170.564,35.673,156.711
C07996=1047.123,98.552,-85.399,170.562,35.672,156.711
C07997=1047.117,98.303,-85.380,170.561,35.670,156.710
C07998=1047.111,98.054,-85.360,170.559,35.668,156.710
C07999=1047.105,97.805,-85.342,170.556,35.667,156.710
C08000=1047.099,97.556,-85.322,170.555,35.665,156.709
C08001=1047.092,97.306,-85.302,170.553,35.664,156.709
C08002=1047.086,97.057,-85.284,170.551,35.662,156.709
C08003=1047.080,96.808,-85.264,170.550,35.660,156.708
C08004=1047.074,96.559,-85.245,170.548,35.659,156.708
C08005=1047.068,96.309,-85.226,170.546,35.657,156.708
C08006=1047.061,96.060,-85.207,170.544,35.656,156.708
C08007=1047.055,95.812,-85.187,170.542,35.654,156.707
C08008=1047.049,95.562,-85.169,170.540,35.652,156.707
C08009=1047.043,95.313,-85.149,170.539,35.651,156.707
C08010=1047.037,95.064,-85.131,170.537,35.649,156.706
C08011=1047.030,94.814,-85.110,170.535,35.647,156.706
C08012=1047.024,94.565,-85.092,170.534,35.646,156.706
C08013=1047.018,94.316,-85.072,170.531,35.644,156.705
C08014=1047.012,94.066,-85.053,170.529,35.642,156.705
C08015=1047.006,93.781,-85.031,170.528,35.641,156.705
C08016=1046.998,93.495,-85.010,170.526,35.639,156.704
C08017=1046.991,93.209,-84.987,170.524,35.637,156.704
C08018=1046.984,92.923,-84.966,170.522,35.634,156.704
C08019=1046.978,92.674,-84.946,170.520,35.633,156.703
C08020=1046.972,92.425,-84.927,170.518,35.631,156.703
C08021=1046.966,92.176,-84.908,170.516,35.630,156.703
C08022=1046.959,91.927,-84.889,170.514,35.628,156.702
C08023=1046.954,91.677,-84.870,170.513,35.626,156.702
C08024=1046.947,91.428,-84.851,170.511,35.625,156.702
C08025=1046.942,91.179,-84.832,170.509,35.623,156.702
C08026=1046.935,90.930,-84.813,170.508,35.621,156.701
C08027=1046.929,90.681,-84.793,170.506,35.620,156.701
C08028=1046.923,90.431,-84.775,170.504,35.618,156.701
C08029=1046.917,90.182,-84.755,170.502,35.616,156.700
C08030=1046.911,89.933,-84.737,170.500,35.614,156.700
C08031=1046.904,89.684,-84.718,170.499,35.613,156.700
C08032=1046.898,89.435,-84.700,170.497,35.611,156.699
C08033=1046.892,89.185,-84.680,170.495,35.609,156.699
C08034=1046.886,88.936,-84.662,170.494,35.608,156.699
C08035=1046.879,88.687,-84.643,170.491,35.606,156.699
C08036=1046.873,88.438,-84.624,170.489,35.605,156.698
C08037=1046.867,88.188,-84.605,170.488,35.603,156.698
C08038=1046.861,87.939,-84.586,170.486,35.602,156.698
C08039=1046.854,87.690,-84.568,170.484,35.600,156.697
C08040=1046.848,87.441,-84.549,170.483,35.599,156.697
C08041=1046.842,87.192,-84.530,170.481,35.597,156.697
C08042=1046.836,86.943,-84.511,170.479,35.595,156.697
C08043=1046.829,86.693,-84.493,170.477,35.593,156.696
C08044=1046.823,86.444,-84.474,170.475,35.592,156.696
C08045=1046.817,86.195,-84.455,170.473,35.590,156.696
C08046=1046.811,85.946,-84.436,170.472,35.589,156.695
C08047=1046.804,85.697,-84.417,170.470,35.587,156.695
C08048=1046.798,85.448,-84.399,170.469,35.586,156.695
C08049=1046.792,85.198,-84.381,170.467,35.584,156.695
C08050=1046.786,84.948,-84.362,170.464,35.582,156.694
C08051=1046.780,84.699,-84.343,170.463,35.581,156.694
C08052=1046.773,84.450,-84.324,170.461,35.579,156.694
C08053=1046.767,84.201,-84.306,170.459,35.578,156.693
C08054=1046.761,83.952,-84.286,170.458,35.576,156.693
C08055=1046.755,83.702,-84.268,170.456,35.574,156.693
C08056=1046.748,83.453,-84.249,170.454,35.572,156.693
C08057=1046.743,83.204,-84.232,170.453,35.571,156.692
C08058=1046.736,82.955,-84.213,170.450,35.569,156.692
C08059=1046.731,82.706,-84.194,170.449,35.567,156.692
C08060=1046.724,82.457,-84.175,170.447,35.566,156.691
C08061=1046.718,82.207,-84.156,170.445,35.564,156.691
C08062=1046.711,81.958,-84.138,170.444,35.563,156.691
C08063=1046.705,81.709,-84.120,170.442,35.561,156.690
C08064=1046.700,81.459,-84.100,170.440,35.560,156.690
C08065=1046.693,81.210,-84.082,170.439,35.558,156.690
C08066=1046.687,80.961,-84.063,170.436,35.557,156.690
C08067=1046.681,80.712,-84.045,170.434,35.555,156.689
C08068=1046.675,80.463,-84.027,170.433,35.553,156.689
C08069=1046.669,80.213,-84.008,170.431,35.551,156.689
C08070=1046.663,79.964,-83.989,170.430,35.550,156.688
C08071=1046.656,79.715,-83.970,170.428,35.548,156.688
C08072=1046.650,79.465,-83.953,170.426,35.546,156.688
C08073=1046.644,79.216,-83.934,170.425,35.544,156.687
C08074=1046.639,78.967,-83.915,170.422,35.543,156.687
C08075=1046.632,78.718,-83.897,170.420,35.541,156.687
C08076=1046.626,78.469,-83.878,170.419,35.540,156.687
C08077=1046.620,78.219,-83.860,170.417,35.538,156.686
C08078=1046.614,77.970,-83.842,170.416,35.537,156.686
C08079=1046.607,77.684,-83.821,170.414,35.535,156.686
C08080=1046.599,77.398,-83.800,170.412,35.533,156.685
C08081=1046.593,77.112,-83.778,170.409,35.531,156.685
C08082=1046.585,76.826,-83.757,170.407,35.529,156.685
C08083=1046.579,76.577,-83.739,170.405,35.528,156.685
C08084=1046.573,76.328,-83.721,170.404,35.526,156.684
C08085=1046.566,76.079,-83.702,170.402,35.525,156.684
C08086=1046.560,75.829,-83.684,170.400,35.523,156.684
C08087=1046.554,75.580,-83.666,170.399,35.521,156.683
C08088=1046.548,75.331,-83.648,170.397,35.520,156.683
C08089=1046.541,75.081,-83.629,170.396,35.518,156.683
C08090=1046.536,74.832,-83.612,170.393,35.516,156.682
C08091=1046.529,74.583,-83.593,170.391,35.515,156.682
C08092=1046.523,74.334,-83.574,170.390,35.513,156.682
C08093=1046.517,74.084,-83.556,170.388,35.512,156.682
C08094=1046.510,73.836,-83.538,170.386,35.511,156.681
C08095=1046.503,73.586,-83.520,170.385,35.509,156.681
C08096=1046.498,73.337,-83.502,170.383,35.507,156.681
C08097=1046.492,73.088,-83.484,170.381,35.505,156.681
C08098=1046.485,72.839,-83.466,170.379,35.504,156.680
C08099=1046.479,72.589,-83.448,170.377,35.502,156.680
C08100=1046.473,72.340,-83.429,170.375,35.501,156.680
C08101=1046.467,72.091,-83.411,170.374,35.499,156.679
C08102=1046.461,71.842,-83.393,170.372,35.498,156.679
C08103=1046.454,71.592,-83.375,170.371,35.496,156.679
C08104=1046.448,71.342,-83.357,170.369,35.495,156.679
C08105=1046.442,71.094,-83.339,170.367,35.493,156.678
C08106=1046.436,70.844,-83.321,170.365,35.491,156.678
C08107=1046.429,70.595,-83.303,170.363,35.489,156.678
C08108=1046.423,70.345,-83.285,170.361,35.488,156.678
C08109=1046.417,70.097,-83.266,170.360,35.486,156.677
C08110=1046.411,69.847,-83.248,170.358,35.485,156.677
C08111=1046.405,69.597,-83.231,170.356,35.483,156.677
C08112=1046.399,69.348,-83.212,170.355,35.482,156.676
C08113=1046.392,69.100,-83.195,170.353,35.480,156.676
C08114=1046.386,68.850,-83.177,170.351,35.479,156.676
C08115=1046.380,68.601,-83.158,170.349,35.477,156.675
C08116=1046.374,68.351,-83.140,170.347,35.475,156.675
C08117=1046.367,68.102,-83.123,170.346,35.474,156.675
C08118=1046.361,67.853,-83.105,170.344,35.472,156.675
C08119=1046.355,67.603,-83.087,170.342,35.471,156.674
C08120=1046.349,67.354,-83.069,170.341,35.469,156.674
C08121=1046.342,67.106,-83.051,170.339,35.468,156.674
C08122=1046.336,66.856,-83.033,170.337,35.466,156.674
C08123=1046.330,66.606,-83.015,170.335,35.464,156.673
C08124=1046.324,66.357,-82.998,170.333,35.463,156.673
C08125=1046.317,66.108,-82.980,170.331,35.461,156.673
C08126=1046.311,65.859,-82.962,170.330,35.460,156.673
C08127=1046.306,65.609,-82.944,170.328,35.458,156.672
C08128=1046.299,65.360,-82.927,170.327,35.457,156.672
C08129=1046.292,65.111,-82.908,170.325,35.455,156.672
C08130=1046.286,64.861,-82.890,170.323,35.454,156.671
C08131=1046.280,64.612,-82.873,170.321,35.452,156.671
C08132=1046.274,64.363,-82.855,170.319,35.450,156.671
C08133=1046.268,64.113,-82.837,170.317,35.449,156.671
C08134=1046.261,63.865,-82.820,170.316,35.447,156.670
C08135=1046.255,63.615,-82.802,170.314,35.446,156.670
C08136=1046.248,63.366,-82.785,170.312,35.445,156.670
C08137=1046.242,63.116,-82.767,170.311,35.443,156.670
C08138=1046.236,62.867,-82.750,170.309,35.441,156.669
C08139=1046.230,62.617,-82.732,170.307,35.440,156.669
C08140=1046.223,62.368,-82.714,170.305,35.438,156.669
C08141=1046.217,62.119,-82.697,170.303,35.437,156.669
C08142=1046.210,61.870,-82.679,170.301,35.436,156.668
C08143=1046.203,61.584,-82.658,170.299,35.434,156.668
C08144=1046.196,61.298,-82.638,170.297,35.432,156.668
C08145=1046.189,61.012,-82.619,170.296,35.430,156.667
C08146=1046.180,60.725,-82.599,170.294,35.428,156.667
C08147=1046.175,60.476,-82.581,170.292,35.427,156.667
C08148=1046.168,60.227,-82.564,170.290,35.426,156.667
C08149=1046.162,59.977,-82.546,170.288,35.424,156.666
C08150=1046.156,59.728,-82.529,170.286,35.423,156.666
C08151=1046.150,59.479,-82.511,170.284,35.421,156.666
C08152=1046.143,59.229,-82.494,170.283,35.419,156.665
C08153=1046.136,58.981,-82.477,170.281,35.418,156.665
C08154=1046.130,58.731,-82.459,170.279,35.417,156.665
C08155=1046.123,58.481,-82.441,170.278,35.415,156.665
C08156=1046.118,58.232,-82.424,170.276,35.414,156.664
C08157=1046.111,57.983,-82.407,170.274,35.412,156.664
C08158=1046.105,57.734,-82.390,170.272,35.410,156.664
C08159=1046.099,57.484,-82.372,170.270,35.409,156.664
C08160=1046.092,57.235,-82.354,170.268,35.408,156.663
C08161=1046.086,56.986,-82.337,170.267,35.406,156.663
C08162=1046.079,56.737,-82.319,170.265,35.405,156.663
C08163=1046.073,56.488,-82.302,170.263,35.403,156.663
C08164=1046.067,56.238,-82.285,170.262,35.401,156.662
C08165=1046.060,55.989,-82.267,170.260,35.400,156.662
C08166=1046.055,55.739,-82.250,170.258,35.399,156.662
C08167=1046.048,55.490,-82.233,170.257,35.397,156.662
C08168=1046.042,55.241,-82.216,170.254,35.396,156.661
C08169=1046.036,54.991,-82.198,170.252,35.394,156.661
C08170=1046.029,54.742,-82.181,170.251,35.392,156.661
C08171=1046.023,54.493,-82.163,170.249,35.391,156.661
C08172=1046.017,54.243,-82.146,170.247,35.389,156.660
C08173=1046.010,53.994,-82.129,170.246,35.388,156.660
C08174=1046.004,53.744,-82.112,170.244,35.387,156.660
C08175=1045.998,53.495,-82.095,170.242,35.385,156.659
C08176=1045.991,53.246,-82.077,170.241,35.383,156.659
C08177=1045.986,52.997,-82.060,170.238,35.382,156.659
C08178=1045.979,52.747,-82.042,170.236,35.380,156.659
C08179=1045.973,52.498,-82.025,170.235,35.379,156.658
C08180=1045.967,52.248,-82.008,170.233,35.377,156.658
C08181=1045.961,52.000,-81.991,170.231,35.376,156.658
C08182=1045.955,51.750,-81.973,170.230,35.374,156.658
C08183=1045.948,51.501,-81.956,170.228,35.372,156.657
C08184=1045.942,51.251,-81.940,170.226,35.371,156.657
C08185=1045.936,51.002,-81.922,170.225,35.370,156.657
C08186=1045.929,50.753,-81.905,170.222,35.368,156.657
C08187=1045.923,50.504,-81.888,170.220,35.366,156.656
C08188=1045.917,50.254,-81.871,170.219,35.365,156.656
C08189=1045.911,50.005,-81.854,170.217,35.363,156.656
C08190=1045.904,49.755,-81.836,170.215,35.362,156.656
C08191=1045.899,49.506,-81.819,170.214,35.360,156.655
C08192=1045.892,49.256,-81.802,170.212,35.359,156.655
C08193=1045.887,49.007,-81.785,170.210,35.357,156.655
C08194=1045.880,48.758,-81.767,170.209,35.356,156.654
C08195=1045.874,48.508,-81.751,170.207,35.354,156.654
C08196=1045.868,48.259,-81.733,170.205,35.352,156.654
C08197=1045.861,48.010,-81.716,170.203,35.351,156.654
C08198=1045.855,47.761,-81.699,170.201,35.350,156.653
C08199=1045.849,47.511,-81.682,170.200,35.348,156.653
C08200=1045.843,47.262,-81.665,170.198,35.346,156.653
C08201=1045.836,47.012,-81.648,170.196,35.345,156.653
C08202=1045.831,46.763,-81.631,170.195,35.343,156.652
C08203=1045.825,46.514,-81.614,170.193,35.342,156.652
C08204=1045.818,46.264,-81.597,170.191,35.340,156.652
C08205=1045.812,46.016,-81.580,170.189,35.339,156.652
C08206=1045.806,45.767,-81.563,170.187,35.337,156.651
C08207=1045.799,45.479,-81.543,170.185,35.335,156.651
C08208=1045.792,45.193,-81.524,170.183,35.334,156.651
C08209=1045.785,44.907,-81.504,170.181,35.332,156.650
C08210=1045.777,44.620,-81.485,170.179,35.330,156.650
C08211=1045.772,44.371,-81.467,170.178,35.328,156.650
C08212=1045.766,44.121,-81.451,170.176,35.327,156.650
C08213=1045.759,43.872,-81.434,170.174,35.325,156.649
C08214=1045.753,43.623,-81.417,170.172,35.324,156.649
C08215=1045.748,43.374,-81.400,170.170,35.322,156.649
C08216=1045.741,43.124,-81.383,170.168,35.321,156.648
C08217=1045.735,42.875,-81.366,170.167,35.319,156.648
C08218=1045.728,42.625,-81.350,170.165,35.318,156.648
C08219=1045.722,42.376,-81.333,170.163,35.316,156.648
C08220=1045.716,42.127,-81.316,170.162,35.315,156.647
C08221=1045.709,41.877,-81.299,170.160,35.313,156.647
C08222=1045.703,41.628,-81.283,170.158,35.312,156.647
C08223=1045.697,41.379,-81.266,170.156,35.310,156.647
C08224=1045.691,41.129,-81.249,170.154,35.309,156.646
C08225=1045.685,40.880,-81.233,170.152,35.308,156.646
C08226=1045.678,40.631,-81.216,170.150,35.306,156.646
C08227=1045.672,40.381,-81.199,170.149,35.304,156.646
C08228=1045.666,40.132,-81.182,170.147,35.303,156.645
C08229=1045.660,39.882,-81.165,170.145,35.301,156.645
C08230=1045.654,39.633,-81.149,170.144,35.300,156.645
C08231=1045.647,39.384,-81.132,170.142,35.299,156.645
C08232=1045.641,39.134,-81.115,170.140,35.297,156.644
C08233=1045.635,38.885,-81.098,170.139,35.295,156.644
C08234=1045.629,38.636,-81.082,170.136,35.294,156.644
C08235=1045.623,38.386,-81.066,170.134,35.293,156.644
C08236=1045.616,38.137,-81.048,170.133,35.291,156.643
C08237=1045.610,37.888,-81.032,170.131,35.289,156.643
C08238=1045.604,37.638,-81.016,170.129,35.288,156.643
C08239=1045.597,37.389,-80.999,170.127,35.287,156.643
C08240=1045.591,37.139,-80.982,170.126,35.285,156.642
C08241=1045.585,36.890,-80.966,170.124,35.284,156.642
C08242=1045.579,36.640,-80.949,170.122,35.282,156.642
C08243=1045.572,36.392,-80.933,170.121,35.281,156.642
C08244=1045.566,36.142,-80.917,170.118,35.280,156.641
C08245=1045.559,35.892,-80.900,170.116,35.278,156.641
C08246=1045.553,35.643,-80.884,170.114,35.276,156.641
C08247=1045.547,35.394,-80.867,170.113,35.275,156.641
C08248=1045.540,35.144,-80.850,170.111,35.274,156.640
C08249=1045.534,34.895,-80.835,170.109,35.272,156.640
C08250=1045.528,34.646,-80.818,170.108,35.271,156.640
C08251=1045.521,34.396,-80.802,170.106,35.269,156.640
C08252=1045.515,34.147,-80.785,170.104,35.268,156.639
C08253=1045.509,33.898,-80.769,170.102,35.267,156.639
C08254=1045.503,33.648,-80.752,170.101,35.265,156.639
C08255=1045.496,33.399,-80.736,170.098,35.264,156.639
C08256=1045.490,33.149,-80.720,170.096,35.262,156.638
C08257=1045.484,32.900,-80.704,170.095,35.261,156.638
C08258=1045.478,32.651,-80.688,170.093,35.259,156.638
C08259=1045.471,32.401,-80.670,170.091,35.258,156.638
C08260=1045.464,32.152,-80.655,170.089,35.257,156.638
C08261=1045.458,31.903,-80.638,170.088,35.255,156.637
C08262=1045.452,31.653,-80.622,170.086,35.254,156.637
C08263=1045.446,31.403,-80.605,170.084,35.252,156.637
C08264=1045.440,31.154,-80.589,170.083,35.251,156.637
C08265=1045.433,30.905,-80.573,170.081,35.250,156.636
C08266=1045.427,30.656,-80.557,170.078,35.248,156.636
C08267=1045.421,30.406,-80.541,170.076,35.246,156.636
C08268=1045.415,30.156,-80.524,170.075,35.245,156.636
C08269=1045.409,29.907,-80.508,170.073,35.244,156.635
C08270=1045.402,29.658,-80.492,170.071,35.242,156.635
C08271=1045.396,29.371,-80.473,170.069,35.240,156.635
C08272=1045.388,29.085,-80.455,170.067,35.239,156.635
C08273=1045.381,28.799,-80.436,170.065,35.237,156.634
C08274=1045.373,28.512,-80.417,170.063,35.235,156.634
C08275=1045.367,28.263,-80.401,170.062,35.234,156.634
C08276=1045.361,28.013,-80.384,170.059,35.233,156.634
C08277=1045.354,27.763,-80.369,170.057,35.231,156.633
C08278=1045.349,27.514,-80.353,170.055,35.230,156.633
C08279=1045.343,27.265,-80.337,170.054,35.229,156.633
C08280=1045.336,27.016,-80.321,170.052,35.227,156.633
C08281=1045.329,26.766,-80.305,170.050,35.225,156.632
C08282=1045.323,26.516,-80.288,170.049,35.224,156.632
C08283=1045.317,26.267,-80.273,170.047,35.223,156.632
C08284=1045.311,26.018,-80.256,170.045,35.221,156.632
C08285=1045.304,25.769,-80.241,170.043,35.220,156.631
C08286=1045.298,25.520,-80.225,170.042,35.219,156.631
C08287=1045.292,25.269,-80.208,170.040,35.218,156.631
C08288=1045.285,25.020,-80.192,170.037,35.216,156.631
C08289=1045.279,24.770,-80.177,170.035,35.214,156.630
C08290=1045.273,24.521,-80.161,170.034,35.213,156.630
C08291=1045.267,24.272,-80.145,170.032,35.212,156.630
C08292=1045.260,24.023,-80.129,170.030,35.210,156.630
C08293=1045.253,23.773,-80.113,170.028,35.209,156.630
C08294=1045.247,23.524,-80.097,170.027,35.208,156.629
C08295=1045.241,23.274,-80.081,170.025,35.206,156.629
C08296=1045.235,23.025,-80.065,170.023,35.205,156.629
C08297=1045.228,22.776,-80.049,170.021,35.204,156.629
C08298=1045.222,22.526,-80.033,170.020,35.202,156.628
C08299=1045.216,22.277,-80.017,170.017,35.200,156.628
C08300=1045.210,22.027,-80.002,170.015,35.199,156.628
C08301=1045.203,21.778,-79.986,170.013,35.198,156.628
C08302=1045.197,21.528,-79.970,170.012,35.197,156.628
C08303=1045.190,21.279,-79.954,170.010,35.195,156.627
C08304=1045.184,21.030,-79.938,170.008,35.194,156.627
C08305=1045.179,20.780,-79.922,170.006,35.193,156.627
C08306=1045.172,20.531,-79.907,170.005,35.191,156.627
C08307=1045.166,20.281,-79.890,170.003,35.189,156.626
C08308=1045.160,20.032,-79.875,170.001,35.188,156.626
C08309=1045.154,19.782,-79.859,169.999,35.187,156.626
C08310=1045.147,19.533,-79.843,169.997,35.185,156.626
C08311=1045.140,19.284,-79.828,169.995,35.184,156.625
C08312=1045.135,19.034,-79.812,169.993,35.183,156.625
C08313=1045.128,18.785,-79.797,169.991,35.181,156.625
C08314=1045.122,18.535,-79.781,169.989,35.180,156.625
C08315=1045.115,18.286,-79.765,169.988,35.179,156.625
C08316=1045.109,18.036,-79.749,169.986,35.177,156.624
C08317=1045.103,17.787,-79.734,169.984,35.176,156.624
C08318=1045.096,17.538,-79.718,169.982,35.175,156.624
C08319=1045.090,17.288,-79.702,169.980,35.173,156.624
C08320=1045.084,17.039,-79.687,169.979,35.172,156.624
C08321=1045.078,16.789,-79.671,169.977,35.171,156.623
C08322=1045.071,16.540,-79.656,169.975,35.170,156.623
C08323=1045.065,16.291,-79.640,169.972,35.168,156.623
C08324=1045.059,16.041,-79.624,169.971,35.166,156.623
C08325=1045.052,15.792,-79.609,169.969,35.165,156.622
C08326=1045.046,15.542,-79.593,169.967,35.164,156.622
C08327=1045.040,15.293,-79.578,169.965,35.162,156.622
C08328=1045.033,15.043,-79.562,169.963,35.161,156.622
C08329=1045.028,14.794,-79.546,169.962,35.160,156.621
C08330=1045.021,14.544,-79.531,169.960,35.158,156.621
C08331=1045.014,14.295,-79.516,169.958,35.157,156.621
C08332=1045.009,14.045,-79.500,169.956,35.156,156.621
C08333=1045.002,13.796,-79.485,169.955,35.154,156.621
C08334=1044.995,13.547,-79.469,169.953,35.153,156.620
C08335=1044.988,13.253,-79.451,169.951,35.152,156.620
C08336=1044.981,12.960,-79.433,169.947,35.150,156.620
C08337=1044.972,12.667,-79.415,169.945,35.148,156.620
C08338=1044.965,12.373,-79.396,169.943,35.147,156.619
C08339=1044.959,12.124,-79.382,169.941,35.146,156.619
C08340=1044.952,11.875,-79.366,169.940,35.144,156.619
C08341=1044.946,11.625,-79.350,169.938,35.143,156.619
C08342=1044.940,11.375,-79.335,169.936,35.142,156.619
C08343=1044.933,11.126,-79.320,169.934,35.141,156.618
C08344=1044.927,10.876,-79.305,169.932,35.140,156.618
C08345=1044.920,10.627,-79.289,169.930,35.138,156.618
C08346=1044.914,10.378,-79.274,169.929,35.137,156.618
C08347=1044.908,10.129,-79.260,169.927,35.136,156.618
C08348=1044.902,9.879,-79.243,169.925,35.134,156.617
C08349=1044.896,9.630,-79.228,169.922,35.133,156.617
C08350=1044.889,9.380,-79.213,169.920,35.132,156.617
C08351=1044.882,9.131,-79.198,169.919,35.130,156.617
C08352=1044.876,8.881,-79.183,169.917,35.129,156.617
C08353=1044.870,8.632,-79.168,169.915,35.128,156.616
C08354=1044.863,8.383,-79.152,169.913,35.126,156.616
C08355=1044.857,8.133,-79.137,169.911,35.126,156.616
C08356=1044.850,7.883,-79.122,169.909,35.124,156.616
C08357=1044.845,7.633,-79.107,169.908,35.123,156.616
C08358=1044.838,7.384,-79.091,169.906,35.122,156.615
C08359=1044.832,7.135,-79.076,169.904,35.120,156.615
C08360=1044.825,6.885,-79.061,169.902,35.119,156.615
C08361=1044.819,6.635,-79.046,169.900,35.118,156.615
C08362=1044.813,6.387,-79.031,169.898,35.116,156.615
C08363=1044.806,6.137,-79.016,169.896,35.115,156.614
C08364=1044.800,5.888,-79.001,169.894,35.114,156.614
C08365=1044.794,5.638,-78.986,169.892,35.113,156.614
C08366=1044.788,5.389,-78.970,169.890,35.111,156.614
C08367=1044.781,5.139,-78.955,169.888,35.110,156.613
C08368=1044.775,4.889,-78.940,169.887,35.109,156.613
C08369=1044.768,4.640,-78.925,169.885,35.108,156.613
C08370=1044.763,4.391,-78.911,169.883,35.107,156.613
C08371=1044.756,4.142,-78.895,169.881,35.105,156.613
C08372=1044.750,3.892,-78.880,169.879,35.104,156.612
C08373=1044.743,3.643,-78.865,169.877,35.102,156.612
C08374=1044.737,3.393,-78.850,169.875,35.101,156.612
C08375=1044.730,3.143,-78.835,169.874,35.100,156.612
C08376=1044.725,2.894,-78.820,169.872,35.099,156.612
C08377=1044.718,2.645,-78.806,169.869,35.097,156.611
C08378=1044.712,2.395,-78.789,169.867,35.096,156.611
C08379=1044.706,2.150,-78.775,169.865,35.095,156.611
C08380=1044.700,1.904,-78.761,169.864,35.093,156.611
C08381=1044.694,1.659,-78.745,169.862,35.093,156.611
C08382=1044.687,1.413,-78.731,169.860,35.091,156.610
C08383=1044.681,1.168,-78.716,169.858,35.090,156.610
C08384=1044.675,0.922,-78.701,169.856,35.089,156.610
C08385=1044.670,0.677,-78.687,169.854,35.087,156.610
C08386=1044.663,0.432,-78.672,169.853,35.086,156.610
C08387=1044.656,0.182,-78.657,169.851,35.085,156.609
C08388=1044.650,-0.067,-78.642,169.849,35.083,156.609
C08389=1044.644,-0.316,-78.628,169.847,35.082,156.609
C08390=1044.638,-0.566,-78.613,169.845,35.081,156.609
C08391=1044.632,-0.816,-78.597,169.842,35.079,156.609
C08392=1044.626,-1.066,-78.582,169.841,35.078,156.608
C08393=1044.620,-1.315,-78.568,169.839,35.077,156.608
C08394=1044.614,-1.564,-78.553,169.837,35.076,156.608
C08395=1044.607,-1.814,-78.538,169.835,35.074,156.608
C08396=1044.601,-2.064,-78.523,169.833,35.073,156.608
C08397=1044.595,-2.313,-78.508,169.831,35.072,156.607
C08398=1044.589,-2.562,-78.493,169.829,35.070,156.607
C08399=1044.582,-2.846,-78.477,169.827,35.069,156.607
C08400=1044.574,-3.129,-78.460,169.825,35.068,156.607
C08401=1044.568,-3.412,-78.443,169.823,35.066,156.606
C08402=1044.561,-3.695,-78.426,169.821,35.064,156.606
C08403=1044.553,-3.945,-78.412,169.819,35.064,156.606
C08404=1044.547,-4.195,-78.397,169.817,35.062,156.606
C08405=1044.542,-4.444,-78.383,169.815,35.061,156.606
C08406=1044.535,-4.693,-78.368,169.812,35.060,156.605
C08407=1044.528,-4.943,-78.353,169.810,35.059,156.605
C08408=1044.522,-5.192,-78.339,169.809,35.058,156.605
C08409=1044.516,-5.441,-78.324,169.807,35.056,156.605
C08410=1044.510,-5.692,-78.310,169.805,35.055,156.605
C08411=1044.503,-5.941,-78.295,169.803,35.054,156.605
C08412=1044.496,-6.191,-78.280,169.801,35.053,156.604
C08413=1044.491,-6.440,-78.266,169.799,35.052,156.604
C08414=1044.483,-6.689,-78.251,169.797,35.050,156.604
C08415=1044.477,-6.939,-78.237,169.795,35.050,156.604
C08416=1044.472,-7.188,-78.223,169.793,35.048,156.604
C08417=1044.465,-7.438,-78.208,169.791,35.047,156.603
C08418=1044.458,-7.687,-78.193,169.790,35.046,156.603
C08419=1044.453,-7.937,-78.179,169.788,35.045,156.603
C08420=1044.446,-8.186,-78.165,169.786,35.044,156.603
C08421=1044.439,-8.436,-78.150,169.784,35.042,156.603
C08422=1044.433,-8.685,-78.136,169.781,35.042,156.603
C08423=1044.427,-8.935,-78.121,169.779,35.040,156.602
C08424=1044.421,-9.185,-78.106,169.777,35.039,156.602
C08425=1044.414,-9.433,-78.092,169.775,35.038,156.602
C08426=1044.408,-9.684,-78.078,169.773,35.037,156.602
C08427=1044.402,-9.933,-78.063,169.771,35.035,156.602
C08428=1044.395,-10.182,-78.049,169.769,35.034,156.602
C08429=1044.389,-10.432,-78.035,169.767,35.033,156.601
C08430=1044.383,-10.682,-78.020,169.766,35.032,156.601
C08431=1044.376,-10.930,-78.006,169.764,35.031,156.601
C08432=1044.370,-11.181,-77.992,169.762,35.029,156.601
C08433=1044.364,-11.430,-77.977,169.760,35.029,156.601
C08434=1044.357,-11.679,-77.963,169.758,35.027,156.600
C08435=1044.351,-11.929,-77.949,169.756,35.026,156.600
C08436=1044.346,-12.178,-77.934,169.754,35.025,156.600
C08437=1044.339,-12.428,-77.919,169.752,35.024,156.600
C08438=1044.333,-12.677,-77.906,169.750,35.023,156.600
C08439=1044.327,-12.927,-77.891,169.747,35.021,156.600
C08440=1044.320,-13.177,-77.877,169.745,35.020,156.599
C08441=1044.314,-13.426,-77.863,169.743,35.019,156.599
C08442=1044.308,-13.676,-77.849,169.741,35.018,156.599
C08443=1044.302,-13.925,-77.834,169.740,35.017,156.599
C08444=1044.295,-14.174,-77.820,169.738,35.016,156.599
C08445=1044.290,-14.424,-77.806,169.736,35.015,156.598
C08446=1044.283,-14.674,-77.791,169.734,35.013,156.598
C08447=1044.276,-14.924,-77.777,169.732,35.012,156.598
C08448=1044.271,-15.173,-77.763,169.730,35.011,156.598
C08449=1044.264,-15.422,-77.749,169.728,35.010,156.598
C08450=1044.258,-15.671,-77.734,169.726,35.008,156.598
C08451=1044.251,-15.921,-77.721,169.724,35.008,156.597
C08452=1044.245,-16.170,-77.706,169.722,35.006,156.597
C08453=1044.239,-16.420,-77.693,169.720,35.006,156.597
C08454=1044.232,-16.671,-77.678,169.718,35.004,156.597
C08455=1044.226,-16.919,-77.664,169.716,35.004,156.597
C08456=1044.219,-17.169,-77.651,169.714,35.002,156.597
C08457=1044.213,-17.418,-77.636,169.711,35.001,156.596
C08458=1044.207,-17.668,-77.622,169.709,35.000,156.596
C08459=1044.201,-17.918,-77.609,169.707,34.999,156.596
C08460=1044.194,-18.167,-77.594,169.705,34.998,156.596
C08461=1044.188,-18.417,-77.580,169.703,34.997,156.596
C08462=1044.181,-18.666,-77.566,169.701,34.996,156.596
C08463=1044.174,-18.948,-77.551,169.699,34.995,156.596
C08464=1044.167,-19.230,-77.535,169.697,34.993,156.595
C08465=1044.160,-19.511,-77.519,169.695,34.992,156.595
C08466=1044.153,-19.793,-77.504,169.692,34.991,156.595
C08467=1044.146,-20.042,-77.489,169.690,34.990,156.595
C08468=1044.140,-20.292,-77.476,169.688,34.989,156.595
C08469=1044.134,-20.542,-77.462,169.686,34.988,156.595
C08470=1044.128,-20.791,-77.447,169.685,34.987,156.594
C08471=1044.121,-21.041,-77.434,169.683,34.986,156.594
C08472=1044.115,-21.290,-77.420,169.681,34.984,156.594
C08473=1044.108,-21.540,-77.405,169.679,34.984,156.594
C08474=1044.102,-21.789,-77.392,169.677,34.982,156.594
C08475=1044.097,-22.039,-77.378,169.675,34.981,156.593
C08476=1044.090,-22.289,-77.365,169.673,34.980,156.593
C08477=1044.083,-22.537,-77.351,169.670,34.979,156.593
C08478=1044.077,-22.788,-77.337,169.668,34.978,156.593
C08479=1044.071,-23.037,-77.323,169.666,34.977,156.593
C08480=1044.065,-23.287,-77.309,169.664,34.976,156.593
C08481=1044.059,-23.536,-77.295,169.662,34.975,156.593
C08482=1044.052,-23.785,-77.282,169.660,34.974,156.592
C08483=1044.046,-24.035,-77.268,169.658,34.973,156.592
C08484=1044.040,-24.285,-77.254,169.656,34.971,156.592
C08485=1044.033,-24.534,-77.241,169.654,34.971,156.592
C08486=1044.028,-24.784,-77.227,169.652,34.969,156.592
C08487=1044.021,-25.033,-77.213,169.650,34.969,156.592
C08488=1044.015,-25.283,-77.199,169.648,34.967,156.591
C08489=1044.009,-25.532,-77.185,169.646,34.967,156.591
C08490=1044.002,-25.782,-77.172,169.644,34.965,156.591
C08491=1043.997,-26.032,-77.158,169.642,34.965,156.591
C08492=1043.990,-26.281,-77.144,169.640,34.963,156.591
C08493=1043.983,-26.530,-77.130,169.638,34.962,156.591
C08494=1043.978,-26.780,-77.116,169.636,34.961,156.591
C08495=1043.972,-27.029,-77.103,169.634,34.960,156.590
C08496=1043.965,-27.279,-77.089,169.632,34.959,156.590
C08497=1043.959,-27.528,-77.076,169.630,34.958,156.590
C08498=1043.952,-27.778,-77.062,169.627,34.957,156.590
C08499=1043.946,-28.028,-77.049,169.625,34.956,156.590
C08500=1043.940,-28.277,-77.035,169.622,34.956,156.590
C08501=1043.933,-28.527,-77.022,169.620,34.954,156.590
C08502=1043.927,-28.777,-77.008,169.618,34.953,156.589
C08503=1043.920,-29.026,-76.995,169.616,34.952,156.589
C08504=1043.914,-29.276,-76.982,169.614,34.951,156.589
C08505=1043.908,-29.525,-76.968,169.612,34.951,156.589
C08506=1043.901,-29.775,-76.955,169.610,34.949,156.589
C08507=1043.895,-30.024,-76.941,169.608,34.949,156.589
C08508=1043.889,-30.274,-76.927,169.606,34.948,156.589
C08509=1043.882,-30.524,-76.914,169.604,34.947,156.588
C08510=1043.876,-30.773,-76.901,169.602,34.946,156.588
C08511=1043.870,-31.022,-76.887,169.600,34.944,156.588
C08512=1043.863,-31.272,-76.874,169.598,34.944,156.588
C08513=1043.857,-31.522,-76.860,169.596,34.943,156.588
C08514=1043.851,-31.771,-76.848,169.594,34.942,156.588
C08515=1043.844,-32.021,-76.834,169.592,34.941,156.588
C08516=1043.838,-32.271,-76.821,169.590,34.940,156.588
C08517=1043.832,-32.520,-76.808,169.588,34.939,156.587
C08518=1043.826,-32.769,-76.794,169.586,34.938,156.587
C08519=1043.820,-33.019,-76.780,169.584,34.937,156.587
C08520=1043.813,-33.269,-76.767,169.582,34.936,156.587
C08521=1043.807,-33.518,-76.754,169.579,34.935,156.587
C08522=1043.800,-33.768,-76.740,169.576,34.934,156.587
C08523=1043.794,-34.018,-76.727,169.574,34.933,156.587
C08524=1043.788,-34.267,-76.714,169.572,34.933,156.586
C08525=1043.782,-34.516,-76.701,169.570,34.931,156.586
C08526=1043.775,-34.766,-76.687,169.568,34.930,156.586
C08527=1043.768,-35.047,-76.673,169.566,34.929,156.586
C08528=1043.761,-35.328,-76.657,169.564,34.928,156.586
C08529=1043.754,-35.608,-76.643,169.561,34.927,156.586
C08530=1043.748,-35.890,-76.628,169.559,34.926,156.586
C08531=1043.742,-36.139,-76.614,169.557,34.926,156.585
C08532=1043.735,-36.388,-76.601,169.555,34.924,156.585
C08533=1043.729,-36.639,-76.588,169.553,34.923,156.585
C08534=1043.723,-36.888,-76.575,169.551,34.922,156.585
C08535=1043.716,-37.138,-76.562,169.549,34.921,156.585
C08536=1043.710,-37.387,-76.548,169.546,34.921,156.585
C08537=1043.704,-37.637,-76.536,169.544,34.919,156.585
C08538=1043.697,-37.887,-76.522,169.542,34.919,156.585
C08539=1043.691,-38.136,-76.509,169.540,34.918,156.584
C08540=1043.685,-38.385,-76.496,169.538,34.916,156.584
C08541=1043.679,-38.635,-76.483,169.536,34.916,156.584
C08542=1043.673,-38.884,-76.470,169.534,34.915,156.584
C08543=1043.666,-39.135,-76.457,169.532,34.914,156.584
C08544=1043.660,-39.384,-76.444,169.530,34.914,156.584
C08545=1043.654,-39.633,-76.430,169.528,34.912,156.584
C08546=1043.647,-39.883,-76.418,169.526,34.912,156.584
C08547=1043.641,-40.132,-76.405,169.523,34.911,156.583
C08548=1043.635,-40.382,-76.392,169.521,34.910,156.583
C08549=1043.628,-40.632,-76.379,169.519,34.909,156.583
C08550=1043.622,-40.881,-76.366,169.516,34.908,156.583
C08551=1043.616,-41.131,-76.354,169.514,34.907,156.583
C08552=1043.609,-41.380,-76.340,169.512,34.907,156.583
C08553=1043.603,-41.630,-76.328,169.510,34.906,156.583
C08554=1043.597,-41.879,-76.315,169.508,34.905,156.583
C08555=1043.590,-42.129,-76.301,169.506,34.904,156.583
C08556=1043.584,-42.379,-76.289,169.503,34.903,156.582
C08557=1043.578,-42.628,-76.276,169.501,34.902,156.582
C08558=1043.572,-42.878,-76.263,169.499,34.901,156.582
C08559=1043.565,-43.127,-76.250,169.497,34.901,156.582
C08560=1043.560,-43.377,-76.237,169.495,34.900,156.582
C08561=1043.553,-43.626,-76.225,169.493,34.899,156.582
C08562=1043.546,-43.877,-76.212,169.491,34.899,156.582
C08563=1043.540,-44.126,-76.199,169.489,34.897,156.582
C08564=1043.534,-44.376,-76.186,169.486,34.896,156.582
C08565=1043.528,-44.625,-76.173,169.484,34.896,156.581
C08566=1043.521,-44.875,-76.161,169.482,34.895,156.581
C08567=1043.515,-45.125,-76.148,169.480,34.894,156.581
C08568=1043.509,-45.374,-76.135,169.478,34.894,156.581
C08569=1043.503,-45.624,-76.122,169.476,34.893,156.581
C08570=1043.496,-45.873,-76.110,169.474,34.892,156.581
C08571=1043.490,-46.123,-76.097,169.472,34.891,156.581
C08572=1043.484,-46.372,-76.084,169.469,34.890,156.581
C08573=1043.478,-46.622,-76.071,169.467,34.889,156.581
C08574=1043.471,-46.871,-76.059,169.465,34.889,156.581
C08575=1043.465,-47.121,-76.046,169.463,34.888,156.580
C08576=1043.459,-47.370,-76.034,169.461,34.887,156.580
C08577=1043.453,-47.620,-76.021,169.459,34.886,156.580
C08578=1043.447,-47.870,-76.007,169.457,34.885,156.580
C08579=1043.440,-48.120,-75.995,169.454,34.884,156.580
C08580=1043.434,-48.369,-75.982,169.452,34.884,156.580
C08581=1043.428,-48.619,-75.970,169.450,34.883,156.580
C08582=1043.421,-48.869,-75.958,169.448,34.882,156.580
C08583=1043.415,-49.119,-75.945,169.446,34.881,156.580
C08584=1043.409,-49.368,-75.932,169.443,34.881,156.579
C08585=1043.403,-49.618,-75.919,169.441,34.880,156.579
C08586=1043.397,-49.867,-75.908,169.438,34.879,156.579
C08587=1043.390,-50.117,-75.894,169.436,34.878,156.579
C08588=1043.384,-50.366,-75.881,169.434,34.877,156.579
C08589=1043.378,-50.616,-75.869,169.432,34.876,156.579
C08590=1043.372,-50.866,-75.857,169.430,34.876,156.579
C08591=1043.365,-51.147,-75.843,169.427,34.875,156.579
C08592=1043.357,-51.428,-75.829,169.425,34.874,156.579
C08593=1043.350,-51.710,-75.815,169.422,34.873,156.579
C08594=1043.343,-51.990,-75.801,169.420,34.873,156.578
C08595=1043.336,-52.240,-75.789,169.418,34.873,156.579
C08596=1043.331,-52.490,-75.777,169.415,34.872,156.578
C08597=1043.324,-52.739,-75.765,169.413,34.871,156.578
C08598=1043.318,-52.989,-75.752,169.411,34.870,156.578
C08599=1043.311,-53.238,-75.740,169.409,34.870,156.578
C08600=1043.304,-53.488,-75.728,169.407,34.869,156.578
C08601=1043.299,-53.738,-75.715,169.404,34.868,156.578
C08602=1043.292,-53.987,-75.703,169.402,34.868,156.578
C08603=1043.286,-54.237,-75.691,169.400,34.867,156.578
C08604=1043.279,-54.487,-75.679,169.398,34.867,156.578
C08605=1043.273,-54.736,-75.667,169.396,34.866,156.578
C08606=1043.267,-54.986,-75.654,169.393,34.865,156.578
C08607=1043.260,-55.236,-75.642,169.391,34.864,156.578
C08608=1043.253,-55.485,-75.630,169.389,34.864,156.577
C08609=1043.248,-55.735,-75.618,169.387,34.864,156.577
C08610=1043.241,-55.985,-75.606,169.385,34.863,156.577
C08611=1043.235,-56.235,-75.593,169.382,34.862,156.577
C08612=1043.228,-56.484,-75.581,169.380,34.861,156.577
C08613=1043.222,-56.734,-75.569,169.378,34.861,156.577
C08614=1043.216,-56.984,-75.557,169.376,34.860,156.577
C08615=1043.209,-57.233,-75.545,169.374,34.860,156.577
C08616=1043.203,-57.482,-75.533,169.371,34.859,156.577
C08617=1043.197,-57.732,-75.521,169.369,34.858,156.577
C08618=1043.191,-57.982,-75.509,169.367,34.858,156.577
C08619=1043.184,-58.231,-75.497,169.365,34.857,156.577
C08620=1043.178,-58.481,-75.484,169.362,34.857,156.577
C08621=1043.171,-58.731,-75.472,169.360,34.856,156.577
C08622=1043.165,-58.981,-75.460,169.358,34.855,156.577
C08623=1043.159,-59.230,-75.448,169.356,34.855,156.576
C08624=1043.153,-59.479,-75.436,169.354,34.854,156.576
C08625=1043.147,-59.729,-75.423,169.351,34.854,156.576
C08626=1043.140,-59.978,-75.411,169.349,34.853,156.576
C08627=1043.134,-60.228,-75.399,169.347,34.852,156.576
C08628=1043.128,-60.478,-75.387,169.345,34.851,156.576
C08629=1043.121,-60.728,-75.376,169.342,34.851,156.576
C08630=1043.115,-60.978,-75.364,169.340,34.851,156.576
C08631=1043.109,-61.227,-75.352,169.338,34.850,156.576
C08632=1043.103,-61.476,-75.340,169.336,34.849,156.576
C08633=1043.096,-61.726,-75.328,169.333,34.848,156.576
C08634=1043.090,-61.976,-75.315,169.331,34.848,156.576
C08635=1043.083,-62.225,-75.303,169.329,34.848,156.576
C08636=1043.078,-62.475,-75.292,169.327,34.847,156.576
C08637=1043.071,-62.725,-75.280,169.325,34.846,156.576
C08638=1043.065,-62.974,-75.268,169.322,34.845,156.575
C08639=1043.059,-63.224,-75.256,169.320,34.845,156.575
C08640=1043.053,-63.473,-75.244,169.318,34.845,156.575
C08641=1043.047,-63.723,-75.232,169.316,34.844,156.575
C08642=1043.040,-63.973,-75.220,169.313,34.843,156.575
C08643=1043.034,-64.222,-75.208,169.311,34.843,156.575
C08644=1043.028,-64.472,-75.196,169.309,34.842,156.575
C08645=1043.022,-64.722,-75.185,169.307,34.841,156.575
C08646=1043.015,-64.971,-75.173,169.303,34.841,156.575
C08647=1043.009,-65.221,-75.161,169.302,34.841,156.575
C08648=1043.003,-65.470,-75.149,169.299,34.840,156.575
C08649=1042.997,-65.720,-75.138,169.297,34.839,156.575
C08650=1042.990,-65.970,-75.126,169.294,34.838,156.575
C08651=1042.984,-66.220,-75.113,169.292,34.838,156.575
C08652=1042.979,-66.469,-75.102,169.290,34.838,156.575
C08653=1042.972,-66.719,-75.090,169.288,34.837,156.575
C08654=1042.965,-66.968,-75.078,169.285,34.836,156.574
C08655=1042.959,-67.251,-75.065,169.283,34.836,156.574
C08656=1042.952,-67.534,-75.052,169.280,34.835,156.574
C08657=1042.945,-67.816,-75.039,169.278,34.834,156.574
C08658=1042.938,-68.099,-75.026,169.275,34.834,156.574
C08659=1042.932,-68.348,-75.013,169.273,34.833,156.574
C08660=1042.926,-68.599,-75.002,169.271,34.833,156.574
C08661=1042.920,-68.847,-74.990,169.268,34.832,156.574
C08662=1042.914,-69.097,-74.978,169.266,34.831,156.574
C08663=1042.908,-69.348,-74.966,169.264,34.831,156.574
C08664=1042.902,-69.596,-74.955,169.262,34.831,156.574
C08665=1042.895,-69.847,-74.944,169.259,34.830,156.574
C08666=1042.889,-70.097,-74.931,169.257,34.830,156.574
C08667=1042.884,-70.346,-74.920,169.255,34.829,156.574
C08668=1042.877,-70.596,-74.908,169.253,34.828,156.574
C08669=1042.871,-70.844,-74.897,169.250,34.828,156.574
C08670=1042.865,-71.095,-74.885,169.248,34.827,156.574
C08671=1042.859,-71.345,-74.873,169.246,34.827,156.574
C08672=1042.853,-71.594,-74.862,169.243,34.826,156.573
C08673=1042.846,-71.844,-74.850,169.241,34.826,156.573
C08674=1042.841,-72.093,-74.839,169.239,34.825,156.573
C08675=1042.835,-72.343,-74.827,169.237,34.824,156.573
C08676=1042.829,-72.592,-74.816,169.234,34.824,156.573
C08677=1042.822,-72.842,-74.804,169.232,34.823,156.573
C08678=1042.816,-73.092,-74.792,169.230,34.823,156.573
C08679=1042.811,-73.341,-74.780,169.228,34.823,156.573
C08680=1042.804,-73.592,-74.769,169.225,34.822,156.573
C08681=1042.798,-73.841,-74.758,169.223,34.822,156.573
C08682=1042.792,-74.091,-74.746,169.221,34.821,156.573
C08683=1042.786,-74.340,-74.735,169.218,34.820,156.573
C08684=1042.779,-74.590,-74.723,169.216,34.820,156.573
C08685=1042.773,-74.840,-74.712,169.214,34.820,156.573
C08686=1042.767,-75.089,-74.701,169.212,34.819,156.573
C08687=1042.761,-75.339,-74.689,169.209,34.819,156.573
C08688=1042.755,-75.588,-74.678,169.207,34.818,156.573
C08689=1042.749,-75.839,-74.667,169.205,34.818,156.573
C08690=1042.743,-76.087,-74.656,169.202,34.818,156.573
C08691=1042.736,-76.338,-74.644,169.200,34.818,156.573
C08692=1042.730,-76.588,-74.633,169.198,34.817,156.573
C08693=1042.724,-76.837,-74.621,169.195,34.817,156.573
C08694=1042.718,-77.087,-74.610,169.193,34.816,156.573
C08695=1042.712,-77.336,-74.599,169.191,34.816,156.573
C08696=1042.705,-77.587,-74.588,169.188,34.816,156.573
C08697=1042.699,-77.835,-74.577,169.186,34.815,156.573
C08698=1042.693,-78.086,-74.565,169.184,34.815,156.573
C08699=1042.687,-78.335,-74.555,169.181,34.814,156.573
C08700=1042.680,-78.585,-74.544,169.179,34.814,156.573
C08701=1042.674,-78.834,-74.532,169.177,34.813,156.572
C08702=1042.668,-79.084,-74.521,169.174,34.813,156.573
C08703=1042.662,-79.334,-74.510,169.172,34.813,156.573
C08704=1042.656,-79.584,-74.499,169.170,34.812,156.572
C08705=1042.650,-79.833,-74.487,169.167,34.812,156.572
C08706=1042.643,-80.083,-74.476,169.165,34.811,156.572
C08707=1042.638,-80.332,-74.465,169.163,34.811,156.572
C08708=1042.631,-80.582,-74.454,169.160,34.811,156.572
C08709=1042.625,-80.832,-74.444,169.158,34.811,156.572
C08710=1042.619,-81.082,-74.432,169.156,34.811,156.572
C08711=1042.612,-81.331,-74.422,169.153,34.810,156.572
C08712=1042.606,-81.581,-74.411,169.151,34.810,156.572
C08713=1042.600,-81.830,-74.399,169.149,34.810,156.572
C08714=1042.593,-82.080,-74.388,169.146,34.810,156.572
C08715=1042.587,-82.330,-74.378,169.144,34.809,156.572
C08716=1042.580,-82.580,-74.366,169.142,34.809,156.572
C08717=1042.575,-82.829,-74.356,169.139,34.809,156.572
C08718=1042.568,-83.079,-74.345,169.137,34.809,156.572
C08719=1042.561,-83.364,-74.333,169.134,34.808,156.572
C08720=1042.553,-83.648,-74.320,169.131,34.808,156.572
C08721=1042.547,-83.933,-74.308,169.129,34.808,156.572
C08722=1042.539,-84.218,-74.296,169.126,34.808,156.572
C08723=1042.534,-84.468,-74.285,169.124,34.808,156.572
C08724=1042.527,-84.718,-74.274,169.121,34.807,156.572
C08725=1042.521,-84.968,-74.263,169.119,34.807,156.572
C08726=1042.514,-85.218,-74.252,169.117,34.807,156.572
C08727=1042.509,-85.467,-74.241,169.114,34.807,156.572
C08728=1042.503,-85.716,-74.230,169.112,34.806,156.572
C08729=1042.496,-85.966,-74.220,169.109,34.806,156.572
C08730=1042.490,-86.216,-74.209,169.107,34.806,156.572
C08731=1042.484,-86.465,-74.198,169.105,34.806,156.572
C08732=1042.477,-86.715,-74.187,169.102,34.805,156.572
C08733=1042.472,-86.965,-74.176,169.100,34.805,156.573
C08734=1042.464,-87.215,-74.166,169.098,34.805,156.573
C08735=1042.459,-87.464,-74.155,169.095,34.804,156.572
C08736=1042.453,-87.714,-74.144,169.093,34.804,156.572
C08737=1042.446,-87.963,-74.133,169.091,34.804,156.573
C08738=1042.440,-88.214,-74.123,169.089,34.804,156.573
C08739=1042.435,-88.463,-74.112,169.087,34.804,156.573
C08740=1042.428,-88.713,-74.102,169.084,34.804,156.573
C08741=1042.422,-88.962,-74.091,169.082,34.804,156.573
C08742=1042.416,-89.212,-74.080,169.080,34.803,156.573
C08743=1042.409,-89.462,-74.069,169.077,34.803,156.573
C08744=1042.403,-89.711,-74.058,169.075,34.803,156.573
C08745=1042.398,-89.961,-74.048,169.072,34.803,156.573
C08746=1042.391,-90.211,-74.038,169.070,34.803,156.573
C08747=1042.385,-90.461,-74.027,169.068,34.803,156.573
C08748=1042.379,-90.710,-74.016,169.065,34.802,156.573
C08749=1042.373,-90.959,-74.006,169.063,34.802,156.573
C08750=1042.367,-91.210,-73.995,169.060,34.802,156.573
C08751=1042.360,-91.459,-73.985,169.058,34.801,156.573
C08752=1042.355,-91.709,-73.974,169.056,34.801,156.573
C08753=1042.348,-91.958,-73.964,169.053,34.801,156.573
C08754=1042.342,-92.208,-73.952,169.051,34.801,156.573
C08755=1042.336,-92.458,-73.942,169.049,34.801,156.573
C08756=1042.330,-92.708,-73.932,169.046,34.801,156.573
C08757=1042.324,-92.957,-73.921,169.044,34.801,156.573
C08758=1042.317,-93.207,-73.910,169.041,34.801,156.573
C08759=1042.312,-93.457,-73.900,169.039,34.801,156.573
C08760=1042.306,-93.707,-73.889,169.037,34.800,156.573
C08761=1042.299,-93.956,-73.879,169.034,34.800,156.573
C08762=1042.293,-94.207,-73.868,169.032,34.800,156.573
C08763=1042.287,-94.456,-73.858,169.029,34.799,156.573
C08764=1042.281,-94.705,-73.847,169.027,34.799,156.573
C08765=1042.276,-94.955,-73.837,169.025,34.799,156.573
C08766=1042.269,-95.204,-73.827,169.022,34.799,156.573
C08767=1042.264,-95.454,-73.816,169.020,34.799,156.573
C08768=1042.257,-95.704,-73.806,169.017,34.799,156.573
C08769=1042.251,-95.954,-73.795,169.015,34.799,156.573
C08770=1042.245,-96.203,-73.785,169.013,34.799,156.573
C08771=1042.239,-96.453,-73.775,169.010,34.799,156.573
C08772=1042.233,-96.703,-73.764,169.008,34.799,156.573
C08773=1042.227,-96.953,-73.754,169.005,34.798,156.573
C08774=1042.221,-97.203,-73.743,169.003,34.798,156.573
C08775=1042.215,-97.453,-73.734,169.001,34.798,156.573
C08776=1042.209,-97.702,-73.723,168.998,34.798,156.573
C08777=1042.202,-97.951,-73.712,168.996,34.798,156.573
C08778=1042.196,-98.201,-73.703,168.993,34.798,156.573
C08779=1042.191,-98.450,-73.692,168.991,34.798,156.573
C08780=1042.184,-98.701,-73.682,168.988,34.798,156.573
C08781=1042.177,-98.950,-73.672,168.986,34.798,156.573
C08782=1042.172,-99.200,-73.662,168.984,34.798,156.573
C08783=1042.165,-99.488,-73.650,168.981,34.798,156.573
C08784=1042.157,-99.774,-73.638,168.978,34.798,156.573
C08785=1042.150,-100.062,-73.626,168.975,34.798,156.574
C08786=1042.143,-100.348,-73.615,168.972,34.798,156.574
C08787=1042.137,-100.598,-73.605,168.970,34.798,156.574
C08788=1042.131,-100.849,-73.595,168.967,34.798,156.574
C08789=1042.125,-101.098,-73.585,168.965,34.798,156.574
C08790=1042.118,-101.347,-73.575,168.963,34.798,156.574
C08791=1042.113,-101.597,-73.564,168.960,34.798,156.574
C08792=1042.107,-101.847,-73.555,168.958,34.798,156.574
C08793=1042.100,-102.097,-73.545,168.955,34.798,156.574
C08794=1042.095,-102.346,-73.534,168.953,34.798,156.574
C08795=1042.088,-102.596,-73.525,168.951,34.798,156.574
C08796=1042.082,-102.845,-73.514,168.949,34.798,156.574
C08797=1042.076,-103.095,-73.505,168.947,34.798,156.574
C08798=1042.070,-103.345,-73.495,168.944,34.798,156.574
C08799=1042.063,-103.595,-73.484,168.942,34.799,156.574
C08800=1042.057,-103.845,-73.474,168.939,34.799,156.574
C08801=1042.052,-104.095,-73.464,168.937,34.798,156.574
C08802=1042.045,-104.344,-73.454,168.934,34.798,156.574
C08803=1042.039,-104.594,-73.444,168.932,34.799,156.575
C08804=1042.033,-104.844,-73.435,168.929,34.799,156.575
C08805=1042.027,-105.094,-73.425,168.927,34.799,156.575
C08806=1042.021,-105.343,-73.414,168.924,34.799,156.575
C08807=1042.015,-105.593,-73.405,168.922,34.799,156.575
C08808=1042.009,-105.842,-73.395,168.920,34.799,156.575
C08809=1042.003,-106.093,-73.385,168.917,34.799,156.575
C08810=1041.997,-106.342,-73.375,168.915,34.799,156.575
C08811=1041.991,-106.591,-73.365,168.912,34.799,156.575
C08812=1041.984,-106.841,-73.356,168.910,34.799,156.575
C08813=1041.978,-107.091,-73.346,168.907,34.799,156.575
C08814=1041.972,-107.341,-73.335,168.905,34.800,156.575
C08815=1041.966,-107.590,-73.326,168.902,34.799,156.575
C08816=1041.960,-107.840,-73.316,168.900,34.800,156.575
C08817=1041.954,-108.090,-73.306,168.897,34.800,156.575
C08818=1041.948,-108.340,-73.297,168.895,34.800,156.575
C08819=1041.942,-108.590,-73.287,168.892,34.800,156.576
C08820=1041.935,-108.839,-73.278,168.890,34.800,156.576
C08821=1041.929,-109.089,-73.267,168.887,34.801,156.576
C08822=1041.923,-109.338,-73.258,168.885,34.801,156.576
C08823=1041.917,-109.588,-73.248,168.883,34.801,156.576
C08824=1041.911,-109.838,-73.238,168.880,34.801,156.576
C08825=1041.905,-110.088,-73.229,168.878,34.801,156.576
C08826=1041.899,-110.338,-73.219,168.875,34.801,156.576
C08827=1041.893,-110.588,-73.209,168.873,34.801,156.576
C08828=1041.887,-110.837,-73.200,168.871,34.802,156.576
C08829=1041.881,-111.087,-73.191,168.869,34.802,156.576
C08830=1041.875,-111.336,-73.181,168.866,34.802,156.576
C08831=1041.869,-111.586,-73.172,168.864,34.802,156.576
C08832=1041.862,-111.836,-73.162,168.861,34.803,156.577
C08833=1041.856,-112.086,-73.152,168.859,34.803,156.577
C08834=1041.850,-112.335,-73.142,168.856,34.803,156.577
C08835=1041.844,-112.585,-73.133,168.854,34.803,156.577
C08836=1041.837,-112.834,-73.123,168.851,34.804,156.577
C08837=1041.832,-113.085,-73.113,168.849,34.804,156.577
C08838=1041.826,-113.334,-73.103,168.846,34.804,156.577
C08839=1041.821,-113.584,-73.095,168.844,34.804,156.577
C08840=1041.814,-113.834,-73.085,168.841,34.804,156.577
C08841=1041.808,-114.084,-73.076,168.839,34.804,156.577
C08842=1041.802,-114.334,-73.066,168.836,34.805,156.577
C08843=1041.796,-114.583,-73.056,168.834,34.805,156.577
C08844=1041.790,-114.833,-73.047,168.831,34.805,156.578
C08845=1041.784,-115.083,-73.037,168.829,34.805,156.578
C08846=1041.777,-115.333,-73.028,168.826,34.806,156.578
C08847=1041.771,-115.618,-73.018,168.823,34.806,156.578
C08848=1041.763,-115.904,-73.006,168.821,34.806,156.578
C08849=1041.756,-116.191,-72.996,168.818,34.807,156.578
C08850=1041.749,-116.477,-72.985,168.815,34.807,156.578
C08851=1041.743,-116.727,-72.976,168.812,34.807,156.578
C08852=1041.738,-116.976,-72.966,168.810,34.808,156.578
C08853=1041.731,-117.226,-72.957,168.807,34.808,156.578
C08854=1041.726,-117.476,-72.948,168.805,34.808,156.578
C08855=1041.719,-117.726,-72.938,168.803,34.809,156.579
C08856=1041.712,-117.976,-72.929,168.801,34.809,156.579
C08857=1041.706,-118.225,-72.920,168.798,34.809,156.579
C08858=1041.701,-118.474,-72.911,168.796,34.809,156.579
C08859=1041.695,-118.725,-72.902,168.793,34.810,156.579
C08860=1041.689,-118.975,-72.892,168.791,34.810,156.579
C08861=1041.683,-119.224,-72.883,168.788,34.810,156.579
C08862=1041.676,-119.474,-72.873,168.786,34.811,156.579
C08863=1041.670,-119.723,-72.865,168.783,34.811,156.579
C08864=1041.664,-119.973,-72.856,168.781,34.811,156.579
C08865=1041.658,-120.223,-72.846,168.778,34.812,156.580
C08866=1041.652,-120.473,-72.837,168.776,34.812,156.580
C08867=1041.647,-120.723,-72.828,168.773,34.812,156.580
C08868=1041.640,-120.973,-72.818,168.771,34.813,156.580
C08869=1041.634,-121.222,-72.809,168.768,34.813,156.580
C08870=1041.627,-121.472,-72.800,168.766,34.813,156.580
C08871=1041.622,-121.722,-72.791,168.763,34.814,156.580
C08872=1041.616,-121.971,-72.782,168.761,34.814,156.580
C08873=1041.610,-122.221,-72.772,168.758,34.815,156.581
C08874=1041.604,-122.472,-72.763,168.756,34.815,156.581
C08875=1041.598,-122.720,-72.755,168.753,34.815,156.581
C08876=1041.591,-122.970,-72.745,168.751,34.816,156.581
C08877=1041.585,-123.221,-72.736,168.748,34.816,156.581
C08878=1041.580,-123.470,-72.727,168.746,34.817,156.581
C08879=1041.574,-123.720,-72.718,168.744,34.817,156.581
C08880=1041.567,-123.970,-72.709,168.741,34.817,156.581
C08881=1041.562,-124.219,-72.700,168.739,34.818,156.581
C08882=1041.556,-124.469,-72.691,168.736,34.818,156.582
C08883=1041.550,-124.719,-72.682,168.734,34.819,156.582
C08884=1041.543,-124.969,-72.674,168.731,34.820,156.582
C08885=1041.537,-125.218,-72.664,168.729,34.819,156.582
C08886=1041.532,-125.469,-72.655,168.726,34.820,156.582
C08887=1041.525,-125.718,-72.647,168.724,34.821,156.582
///RCONF 1,0,0,0,1,0,0,0,0,0,0,0,0,0,0,0,0,0,0,0,0,0,0,0
C08888=1041.519,-125.968,-72.638,168.721,34.821,156.582
C08889=1041.513,-126.218,-72.628,168.719,34.822,156.582
C08890=1041.507,-126.468,-72.620,168.716,34.822,156.583
C08891=1041.501,-126.717,-72.611,168.714,34.823,156.583
C08892=1041.495,-126.967,-72.602,168.711,34.823,156.583
C08893=1041.488,-127.217,-72.593,168.708,34.824,156.583
C08894=1041.483,-127.466,-72.585,168.706,34.824,156.583
C08895=1041.477,-127.716,-72.575,168.703,34.825,156.583
C08896=1041.471,-127.965,-72.566,168.701,34.825,156.583
C08897=1041.467,-128.215,-72.557,168.699,34.825,156.583
C08898=1041.463,-128.465,-72.546,168.696,34.824,156.583
C08899=1041.459,-128.715,-72.535,168.694,34.823,156.583
C08900=1041.457,-128.965,-72.524,168.692,34.821,156.583
C08901=1041.455,-129.215,-72.511,168.691,34.820,156.583
C08902=1041.454,-129.465,-72.499,168.689,34.817,156.582
C08903=1041.454,-129.715,-72.485,168.687,34.814,156.582
C08904=1041.456,-129.965,-72.472,168.686,34.810,156.581
C08905=1041.458,-130.215,-72.457,168.685,34.807,156.581
C08906=1041.461,-130.465,-72.442,168.683,34.802,156.580
C08907=1041.464,-130.716,-72.427,168.682,34.798,156.579
C08908=1041.468,-130.966,-72.410,168.681,34.793,156.578
C08909=1041.473,-131.216,-72.393,168.680,34.787,156.577
C08910=1041.480,-131.466,-72.376,168.679,34.781,156.576
C08911=1041.131,-131.490,-72.630,168.631,34.973,156.610
C08912=1041.125,-131.240,-72.649,168.633,34.979,156.611
C08913=1041.120,-130.990,-72.665,168.634,34.985,156.611
C08914=1041.115,-130.739,-72.682,168.634,34.990,156.612
C08915=1041.112,-130.489,-72.697,168.636,34.995,156.613
C08916=1041.109,-130.240,-72.713,168.638,34.999,156.614
C08917=1041.108,-129.989,-72.728,168.639,35.003,156.615
C08918=1041.106,-129.739,-72.741,168.640,35.006,156.615
C08919=1041.106,-129.489,-72.755,168.642,35.009,156.615
C08920=1041.107,-129.239,-72.767,168.643,35.012,156.616
C08921=1041.108,-128.989,-72.780,168.646,35.014,156.616
C08922=1041.111,-128.739,-72.791,168.648,35.015,156.616
C08923=1041.114,-128.489,-72.802,168.650,35.016,156.617
C08924=1041.118,-128.239,-72.813,168.652,35.017,156.617
C08925=1041.122,-127.989,-72.822,168.655,35.017,156.617
C08926=1041.128,-127.740,-72.832,168.657,35.017,156.617
C08927=1041.134,-127.491,-72.840,168.660,35.016,156.616
C08928=1041.140,-127.241,-72.849,168.661,35.016,156.616
C08929=1041.146,-126.991,-72.859,168.664,35.015,156.616
C08930=1041.152,-126.742,-72.866,168.666,35.014,156.616
C08931=1041.158,-126.492,-72.876,168.669,35.014,156.616
C08932=1041.164,-126.241,-72.885,168.671,35.014,156.616
C08933=1041.170,-125.993,-72.893,168.674,35.013,156.616
C08934=1041.176,-125.742,-72.902,168.677,35.013,156.616
C08935=1041.183,-125.492,-72.912,168.679,35.012,156.615
C08936=1041.189,-125.243,-72.920,168.682,35.012,156.615
C08937=1041.195,-124.993,-72.929,168.684,35.011,156.615
C08938=1041.201,-124.743,-72.938,168.687,35.011,156.615
C08939=1041.207,-124.494,-72.947,168.689,35.010,156.615
C08940=1041.213,-124.244,-72.956,168.692,35.010,156.615
C08941=1041.219,-123.994,-72.965,168.694,35.009,156.615
///RCONF 1,0,0,0,0,0,0,0,0,0,0,0,0,0,0,0,0,0,0,0,0,0,0,0
C08942=1041.225,-123.743,-72.974,168.697,35.009,156.615
C08943=1041.230,-123.494,-72.983,168.699,35.009,156.614
C08944=1041.237,-123.245,-72.992,168.702,35.008,156.614
C08945=1041.243,-122.994,-73.001,168.705,35.008,156.614
C08946=1041.249,-122.745,-73.010,168.707,35.007,156.614
C08947=1041.255,-122.495,-73.020,168.710,35.006,156.614
C08948=1041.261,-122.245,-73.029,168.712,35.007,156.614
C08949=1041.268,-121.995,-73.038,168.714,35.006,156.614
C08950=1041.273,-121.746,-73.047,168.716,35.005,156.614
C08951=1041.279,-121.496,-73.056,168.719,35.005,156.614
C08952=1041.285,-121.246,-73.065,168.721,35.004,156.613
C08953=1041.291,-120.997,-73.075,168.724,35.004,156.613
C08954=1041.297,-120.747,-73.083,168.726,35.004,156.613
C08955=1041.304,-120.497,-73.092,168.729,35.003,156.613
C08956=1041.310,-120.247,-73.102,168.731,35.003,156.613
C08957=1041.315,-119.998,-73.110,168.734,35.003,156.613
C08958=1041.321,-119.748,-73.120,168.736,35.002,156.613
C08959=1041.327,-119.498,-73.130,168.739,35.002,156.613
C08960=1041.334,-119.248,-73.139,168.742,35.001,156.613
C08961=1041.340,-118.998,-73.147,168.744,35.001,156.612
C08962=1041.346,-118.749,-73.157,168.747,35.001,156.612
C08963=1041.352,-118.499,-73.166,168.749,35.000,156.612
C08964=1041.358,-118.249,-73.176,168.752,35.000,156.612
C08965=1041.364,-118.000,-73.185,168.754,35.000,156.612
C08966=1041.370,-117.749,-73.194,168.757,34.999,156.612
C08967=1041.376,-117.500,-73.203,168.759,34.999,156.612
C08968=1041.382,-117.250,-73.213,168.762,34.999,156.612
C08969=1041.388,-117.001,-73.222,168.764,34.998,156.612
C08970=1041.394,-116.751,-73.232,168.767,34.998,156.612
C08971=1041.401,-116.501,-73.240,168.769,34.998,156.611
C08972=1041.407,-116.215,-73.251,168.771,34.997,156.611
C08973=1041.414,-115.929,-73.262,168.774,34.997,156.611
C08974=1041.421,-115.642,-73.273,168.777,34.997,156.611
C08975=1041.428,-115.357,-73.284,168.780,34.996,156.611
C08976=1041.434,-115.106,-73.293,168.782,34.996,156.611
C08977=1041.440,-114.856,-73.303,168.785,34.996,156.611
C08978=1041.447,-114.606,-73.312,168.787,34.995,156.611
C08979=1041.452,-114.357,-73.321,168.790,34.995,156.611
C08980=1041.458,-114.108,-73.331,168.792,34.995,156.611
C08981=1041.464,-113.858,-73.341,168.795,34.994,156.610
C08982=1041.471,-113.608,-73.350,168.797,34.994,156.610
C08983=1041.477,-113.358,-73.360,168.800,34.994,156.610
C08984=1041.483,-113.108,-73.369,168.802,34.994,156.610
C08985=1041.489,-112.859,-73.379,168.805,34.993,156.610
C08986=1041.495,-112.609,-73.388,168.807,34.994,156.610
C08987=1041.501,-112.360,-73.398,168.810,34.993,156.610
C08988=1041.507,-112.110,-73.407,168.812,34.993,156.610
C08989=1041.513,-111.860,-73.417,168.815,34.993,156.610
C08990=1041.519,-111.610,-73.426,168.817,34.993,156.610
C08991=1041.526,-111.361,-73.436,168.820,34.992,156.610
C08992=1041.532,-111.111,-73.445,168.822,34.992,156.610
C08993=1041.538,-110.861,-73.455,168.825,34.992,156.609
C08994=1041.544,-110.611,-73.465,168.827,34.992,156.609
C08995=1041.550,-110.361,-73.475,168.830,34.991,156.609
C08996=1041.556,-110.111,-73.484,168.832,34.991,156.609
C08997=1041.562,-109.861,-73.494,168.835,34.991,156.609
C08998=1041.568,-109.612,-73.503,168.837,34.991,156.609
C08999=1041.575,-109.362,-73.514,168.839,34.990,156.609
C09000=1041.581,-109.113,-73.523,168.841,34.990,156.609
C09001=1041.587,-108.863,-73.533,168.844,34.990,156.609
C09002=1041.593,-108.613,-73.542,168.846,34.990,156.609
C09003=1041.599,-108.363,-73.552,168.849,34.989,156.609
C09004=1041.605,-108.113,-73.562,168.851,34.989,156.609
C09005=1041.612,-107.864,-73.571,168.854,34.989,156.609
C09006=1041.618,-107.614,-73.581,168.856,34.989,156.609
C09007=1041.623,-107.364,-73.592,168.859,34.989,156.608
C09008=1041.629,-107.115,-73.601,168.861,34.989,156.608
C09009=1041.635,-106.865,-73.610,168.864,34.989,156.608
C09010=1041.641,-106.616,-73.620,168.866,34.988,156.608
C09011=1041.648,-106.367,-73.630,168.869,34.988,156.608
C09012=1041.653,-106.116,-73.640,168.871,34.988,156.608
C09013=1041.659,-105.867,-73.650,168.874,34.988,156.608
C09014=1041.666,-105.616,-73.660,168.876,34.988,156.608
C09015=1041.673,-105.367,-73.670,168.879,34.988,156.608
C09016=1041.678,-105.117,-73.680,168.881,34.987,156.608
C09017=1041.684,-104.867,-73.690,168.883,34.988,156.608
C09018=1041.691,-104.617,-73.699,168.886,34.988,156.608
C09019=1041.697,-104.368,-73.710,168.888,34.987,156.608
C09020=1041.702,-104.118,-73.720,168.891,34.987,156.608
C09021=1041.709,-103.868,-73.729,168.893,34.987,156.608
C09022=1041.715,-103.619,-73.740,168.896,34.987,156.608
C09023=1041.721,-103.369,-73.749,168.898,34.987,156.607
C09024=1041.727,-103.119,-73.759,168.901,34.987,156.607
C09025=1041.733,-102.870,-73.770,168.903,34.987,156.607
C09026=1041.739,-102.620,-73.779,168.906,34.987,156.607
C09027=1041.745,-102.370,-73.789,168.908,34.987,156.607
C09028=1041.751,-102.121,-73.800,168.911,34.987,156.607
C09029=1041.757,-101.871,-73.809,168.913,34.987,156.607
C09030=1041.763,-101.621,-73.819,168.915,34.986,156.607
C09031=1041.769,-101.372,-73.830,168.918,34.986,156.607
C09032=1041.776,-101.121,-73.840,168.920,34.986,156.607
C09033=1041.782,-100.872,-73.851,168.922,34.987,156.607
C09034=1041.788,-100.622,-73.860,168.924,34.987,156.607
C09035=1041.794,-100.373,-73.870,168.927,34.986,156.607
C09036=1041.802,-100.085,-73.882,168.930,34.986,156.607
C09037=1041.808,-99.798,-73.893,168.932,34.986,156.607
C09038=1041.816,-99.511,-73.905,168.935,34.986,156.607
C09039=1041.822,-99.224,-73.917,168.938,34.986,156.607
C09040=1041.829,-98.974,-73.927,168.940,34.986,156.607
C09041=1041.835,-98.724,-73.937,168.943,34.986,156.607
C09042=1041.841,-98.474,-73.947,168.945,34.986,156.607
C09043=1041.847,-98.225,-73.958,168.948,34.986,156.607
C09044=1041.853,-97.975,-73.967,168.950,34.986,156.606
C09045=1041.859,-97.726,-73.978,168.953,34.986,156.606
